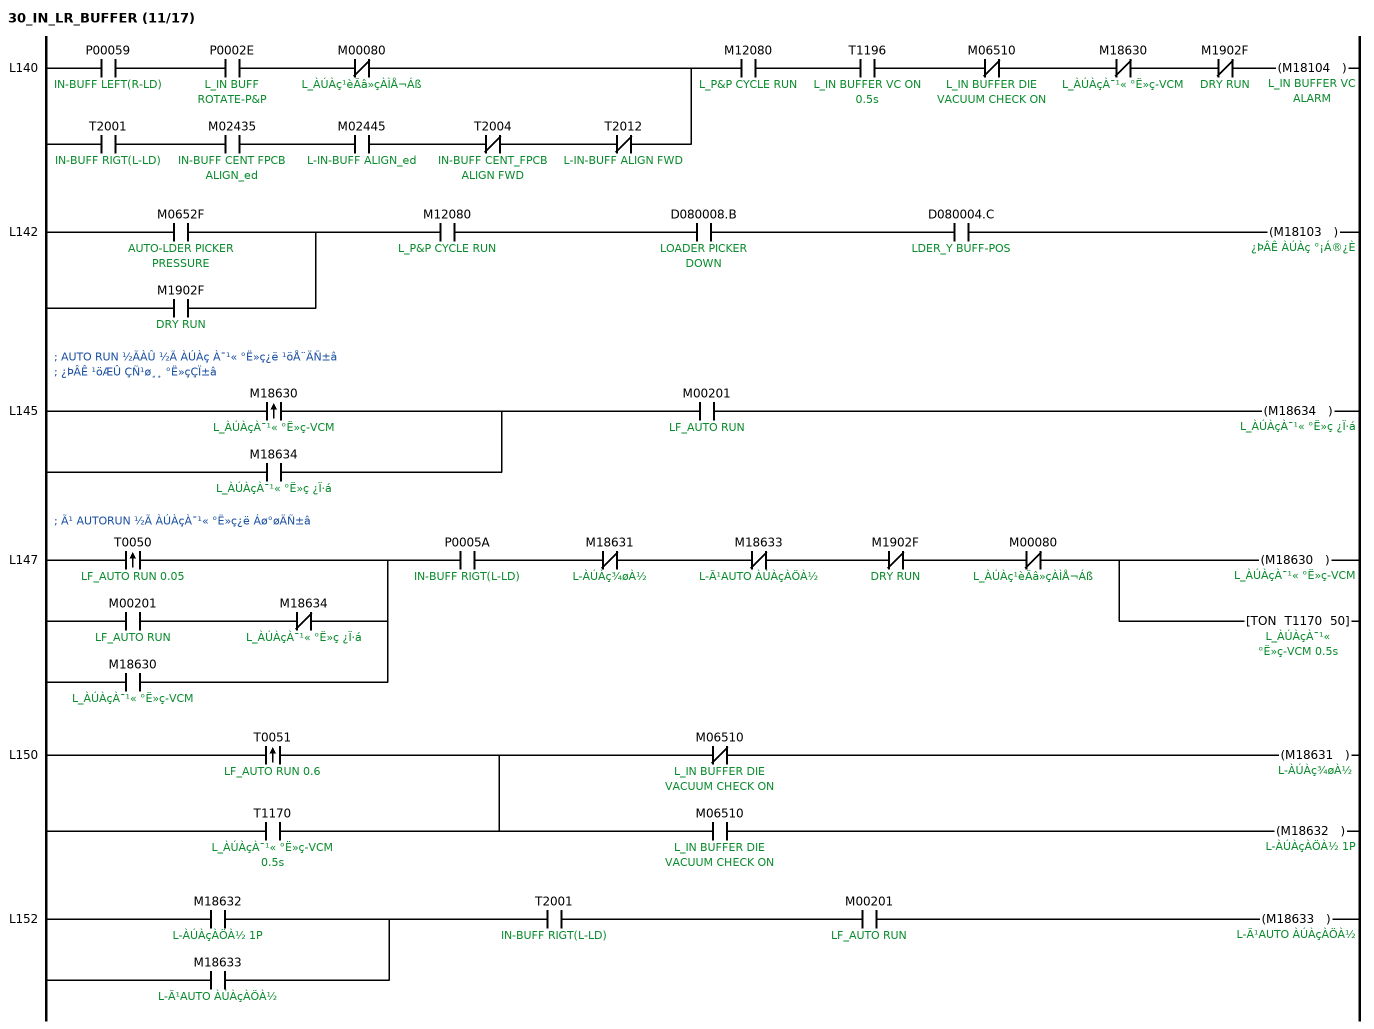
[picture p216: 30_IN_LR_BUFFER rungs L140-L152]
; L140
LOAD      P00059	// IN-BUFF LEFT(R-LD)
AND       P0002E	// L_IN BUFF ROTATE-P&P
AND NOT   M00080	// L_ÀÚÀç¹èÃâ»çÀÌÅ¬Áß
LOAD      T2001	// IN-BUFF RIGT(L-LD)
AND       M02435	// IN-BUFF CENT FPCB ALIGN_ed
AND       M02445	// L-IN-BUFF ALIGN_ed
AND NOT   T2004	// IN-BUFF CENT_FPCB ALIGN FWD
AND NOT   T2012	// L-IN-BUFF ALIGN FWD
OR LOAD
AND       M12080	// L_P&P CYCLE RUN
AND       T1196	// L_IN BUFFER VC ON 0.5s
AND NOT   M06510	// L_IN BUFFER DIE VACUUM CHECK ON
AND NOT   M18630	// L_ÀÚÀçÀ¯¹« °Ë»ç-VCM
AND NOT   M1902F	// DRY RUN
OUT       M18104	// L_IN BUFFER VC ALARM
; L142
LOAD      M0652F	// AUTO-LDER PICKER PRESSURE
OR        M1902F	// DRY RUN
AND       M12080	// L_P&P CYCLE RUN
AND       D080008.B	// LOADER PICKER DOWN
AND       D080004.C	// LDER_Y BUFF-POS
OUT       M18103	// ¿ÞÂÊ ÀÚÀç °¡Á®¿È
// AUTO RUN ½ÃÀÛ ½Ã ÀÚÀç À¯¹« °Ë»ç¿ë ¹öÅ¨ÄÑ±â
; L145
LOADP     M18630	// L_ÀÚÀçÀ¯¹« °Ë»ç-VCM
OR        M18634	// L_ÀÚÀçÀ¯¹« °Ë»ç ¿Ï·á
AND       M00201	// LF_AUTO RUN
OUT       M18634	// L_ÀÚÀçÀ¯¹« °Ë»ç ¿Ï·á
// output comment: ¿ÞÂÊ ¹öÆÛ ÇÑ¹ø¸¸ °Ë»çÇÏ±â
; L147
LOADP     T0050	// LF_AUTO RUN 0.05
LOAD      M00201	// LF_AUTO RUN
AND NOT   M18634	// L_ÀÚÀçÀ¯¹« °Ë»ç ¿Ï·á
OR LOAD
OR        M18630	// L_ÀÚÀçÀ¯¹« °Ë»ç-VCM
AND       P0005A	// IN-BUFF RIGT(L-LD)
AND NOT   M18631	// L-ÀÚÀç¾øÀ½
AND NOT   M18633	// L-Ã¹AUTO ÀÚÀçÀÖÀ½
AND NOT   M1902F	// DRY RUN
AND NOT   M00080	// L_ÀÚÀç¹èÃâ»çÀÌÅ¬Áß
OUT       M18630	// L_ÀÚÀçÀ¯¹« °Ë»ç-VCM
TON       T1170 50	// L_ÀÚÀçÀ¯¹« °Ë»ç-VCM 0.5s
// output comment: Ã¹ AUTORUN ½Ã ÀÚÀçÀ¯¹« °Ë»ç¿ë Áø°øÄÑ±â
; L150
LOADP     T0051	// LF_AUTO RUN 0.6
OR        T1170	// L_ÀÚÀçÀ¯¹« °Ë»ç-VCM 0.5s
MPUSH
AND NOT   M06510	// L_IN BUFFER DIE VACUUM CHECK ON
OUT       M18631	// L-ÀÚÀç¾øÀ½
MPOP
AND       M06510	// L_IN BUFFER DIE VACUUM CHECK ON
OUT       M18632	// L-ÀÚÀçÀÖÀ½ 1P
; L152
LOAD      M18632	// L-ÀÚÀçÀÖÀ½ 1P
OR        M18633	// L-Ã¹AUTO ÀÚÀçÀÖÀ½
AND       T2001	// IN-BUFF RIGT(L-LD)
AND       M00201	// LF_AUTO RUN
OUT       M18633	// L-Ã¹AUTO ÀÚÀçÀÖÀ½

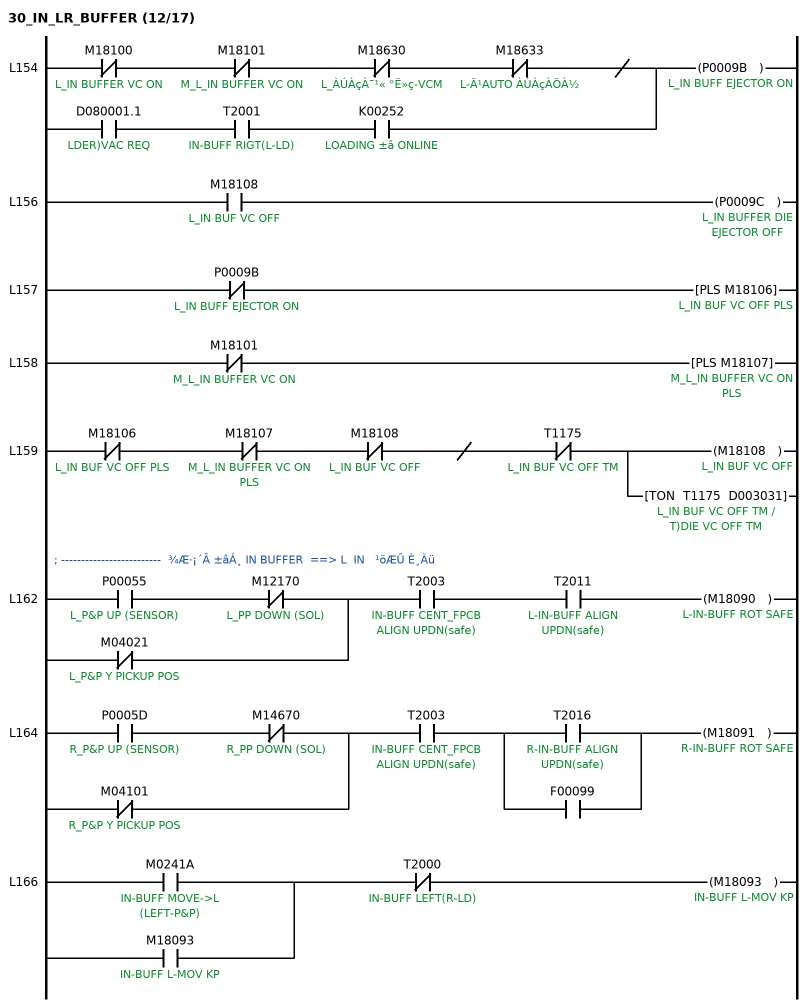
; L154
LOAD NOT  M18100	// L_IN BUFFER VC ON
AND NOT   M18101	// M_L_IN BUFFER VC ON
AND NOT   M18630	// L_ÀÚÀçÀ¯¹« °Ë»ç-VCM
AND NOT   M18633	// L-Ã¹AUTO ÀÚÀçÀÖÀ½
NOT
LOAD      D080001.1	// LDER)VAC REQ
AND       T2001	// IN-BUFF RIGT(L-LD)
AND       K00252	// LOADING ±â ONLINE
OR LOAD
OUT       P0009B	// L_IN BUFF EJECTOR ON
; L156
LOAD      M18108	// L_IN BUF VC OFF
OUT       P0009C	// L_IN BUFFER DIE EJECTOR OFF
; L157
LOAD NOT  P0009B	// L_IN BUFF EJECTOR ON
OUTP      M18106	// L_IN BUF VC OFF PLS
; L158
LOAD NOT  M18101	// M_L_IN BUFFER VC ON
OUTP      M18107	// M_L_IN BUFFER VC ON PLS
; L159
LOAD NOT  M18106	// L_IN BUF VC OFF PLS
AND NOT   M18107	// M_L_IN BUFFER VC ON PLS
AND NOT   M18108	// L_IN BUF VC OFF
NOT
AND NOT   T1175	// L_IN BUF VC OFF TM
OUT       M18108	// L_IN BUF VC OFF
TON       T1175 D003031	// L_IN BUF VC OFF TM / T)DIE VC OFF TM
// -------------------------  ¾Æ·¡´Â ±âÁ¸ IN BUFFER  ==> L  IN   ¹öÆÛ È¸Àü
; L162
LOAD      P00055	// L_P&P UP (SENSOR)
AND NOT   M12170	// L_PP DOWN (SOL)
OR NOT    M04021	// L_P&P Y PICKUP POS
AND       T2003	// IN-BUFF CENT_FPCB ALIGN UPDN(safe)
AND       T2011	// L-IN-BUFF ALIGN UPDN(safe)
OUT       M18090	// L-IN-BUFF ROT SAFE
; L164
LOAD      P0005D	// R_P&P UP (SENSOR)
AND NOT   M14670	// R_PP DOWN (SOL)
OR NOT    M04101	// R_P&P Y PICKUP POS
AND       T2003	// IN-BUFF CENT_FPCB ALIGN UPDN(safe)
LOAD      T2016	// R-IN-BUFF ALIGN UPDN(safe)
OR        F00099
AND LOAD
OUT       M18091	// R-IN-BUFF ROT SAFE
; L166
LOAD      M0241A	// IN-BUFF MOVE->L (LEFT-P&P)
OR        M18093	// IN-BUFF L-MOV KP
AND NOT   T2000	// IN-BUFF LEFT(R-LD)
OUT       M18093	// IN-BUFF L-MOV KP

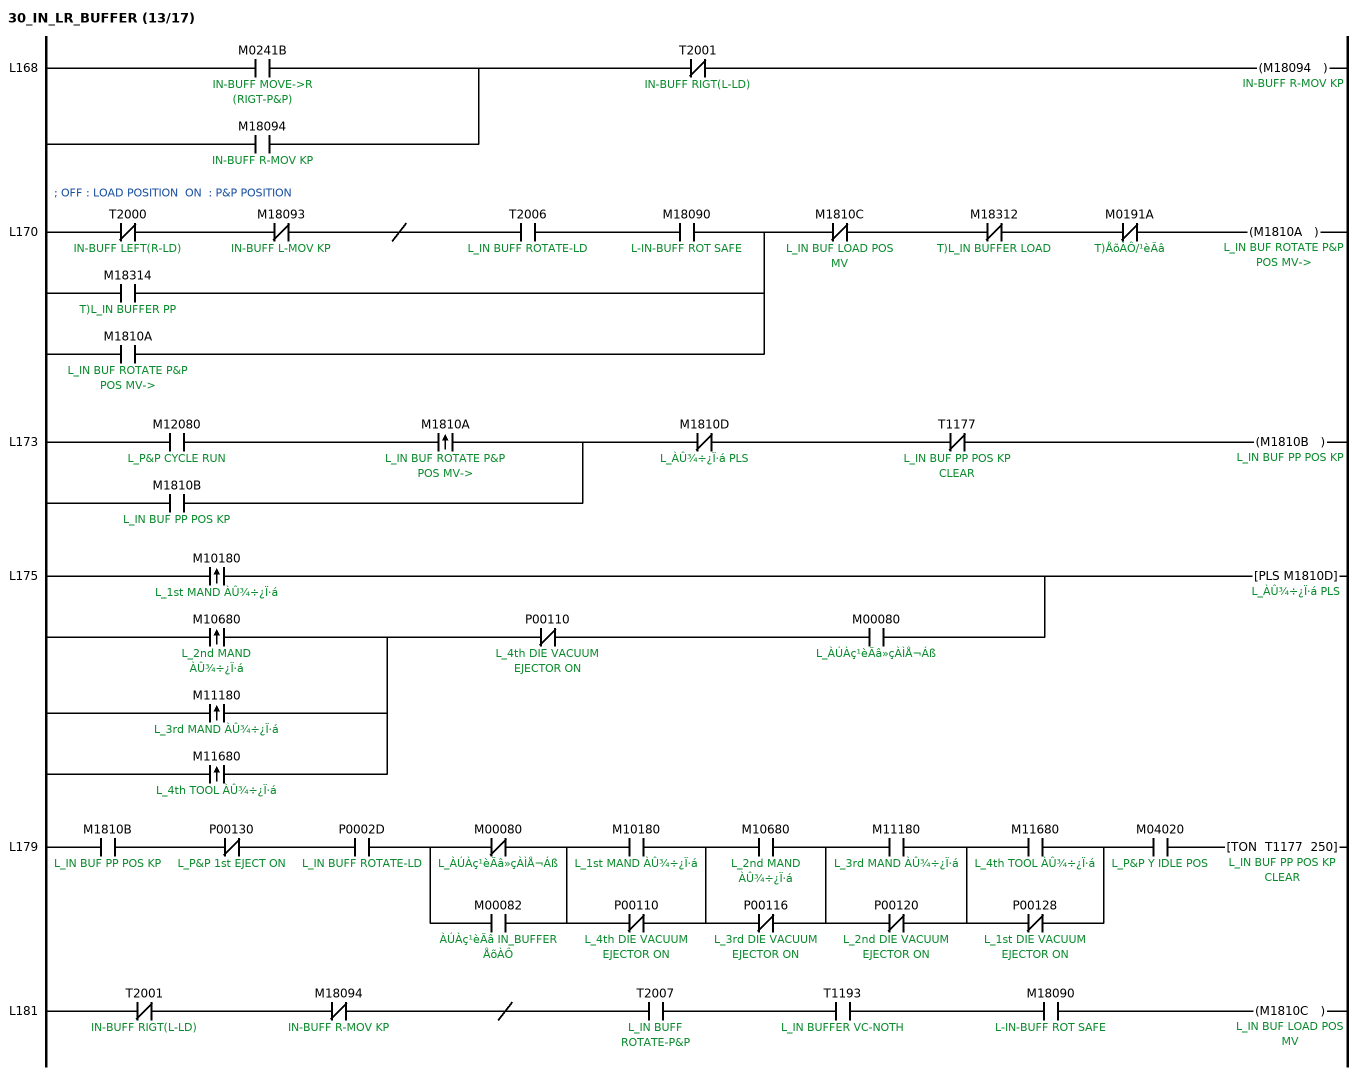
; L168
LOAD      M0241B	// IN-BUFF MOVE->R (RIGT-P&P)
OR        M18094	// IN-BUFF R-MOV KP
AND NOT   T2001	// IN-BUFF RIGT(L-LD)
OUT       M18094	// IN-BUFF R-MOV KP
; L170
LOAD NOT  T2000	// IN-BUFF LEFT(R-LD)
AND NOT   M18093	// IN-BUFF L-MOV KP
NOT
AND       T2006	// L_IN BUFF ROTATE-LD
AND       M18090	// L-IN-BUFF ROT SAFE
OR        M18314	// T)L_IN BUFFER PP
OR        M1810A	// L_IN BUF ROTATE P&P POS MV->
AND NOT   M1810C	// L_IN BUF LOAD POS MV
AND NOT   M18312	// T)L_IN BUFFER LOAD
AND NOT   M0191A	// T)ÅõÀÔ/¹èÃâ
OUT       M1810A	// L_IN BUF ROTATE P&P POS MV->
// output comment: OFF : LOAD POSITION  ON  : P&P POSITION
; L173
LOAD      M12080	// L_P&P CYCLE RUN
ANDP      M1810A	// L_IN BUF ROTATE P&P POS MV->
OR        M1810B	// L_IN BUF PP POS KP
AND NOT   M1810D	// L_ÀÛ¾÷¿Ï·á PLS
AND NOT   T1177	// L_IN BUF PP POS KP CLEAR
OUT       M1810B	// L_IN BUF PP POS KP
; L175
LOADP     M10180	// L_1st MAND ÀÛ¾÷¿Ï·á
LOADP     M10680	// L_2nd MAND ÀÛ¾÷¿Ï·á
ORP       M11180	// L_3rd MAND ÀÛ¾÷¿Ï·á
ORP       M11680	// L_4th TOOL ÀÛ¾÷¿Ï·á
AND NOT   P00110	// L_4th DIE VACUUM EJECTOR ON
AND       M00080	// L_ÀÚÀç¹èÃâ»çÀÌÅ¬Áß
OR LOAD
OUTP      M1810D	// L_ÀÛ¾÷¿Ï·á PLS
; L179
LOAD      M1810B	// L_IN BUF PP POS KP
AND NOT   P00130	// L_P&P 1st EJECT ON
AND       P0002D	// L_IN BUFF ROTATE-LD
LOAD NOT  M00080	// L_ÀÚÀç¹èÃâ»çÀÌÅ¬Áß
OR        M00082	// ÀÚÀç¹èÃâ IN_BUFFER ÅõÀÔ 
AND LOAD
LOAD      M10180	// L_1st MAND ÀÛ¾÷¿Ï·á
OR NOT    P00110	// L_4th DIE VACUUM EJECTOR ON
AND LOAD
LOAD      M10680	// L_2nd MAND ÀÛ¾÷¿Ï·á
OR NOT    P00116	// L_3rd DIE VACUUM EJECTOR ON
AND LOAD
LOAD      M11180	// L_3rd MAND ÀÛ¾÷¿Ï·á
OR NOT    P00120	// L_2nd DIE VACUUM EJECTOR ON
AND LOAD
LOAD      M11680	// L_4th TOOL ÀÛ¾÷¿Ï·á
OR NOT    P00128	// L_1st DIE VACUUM EJECTOR ON
AND LOAD
AND       M04020	// L_P&P Y IDLE POS
TON       T1177 250	// L_IN BUF PP POS KP CLEAR
; L181
LOAD NOT  T2001	// IN-BUFF RIGT(L-LD)
AND NOT   M18094	// IN-BUFF R-MOV KP
NOT
AND       T2007	// L_IN BUFF ROTATE-P&P
AND       T1193	// L_IN BUFFER VC-NOTH
AND       M18090	// L-IN-BUFF ROT SAFE
OUT       M1810C	// L_IN BUF LOAD POS MV

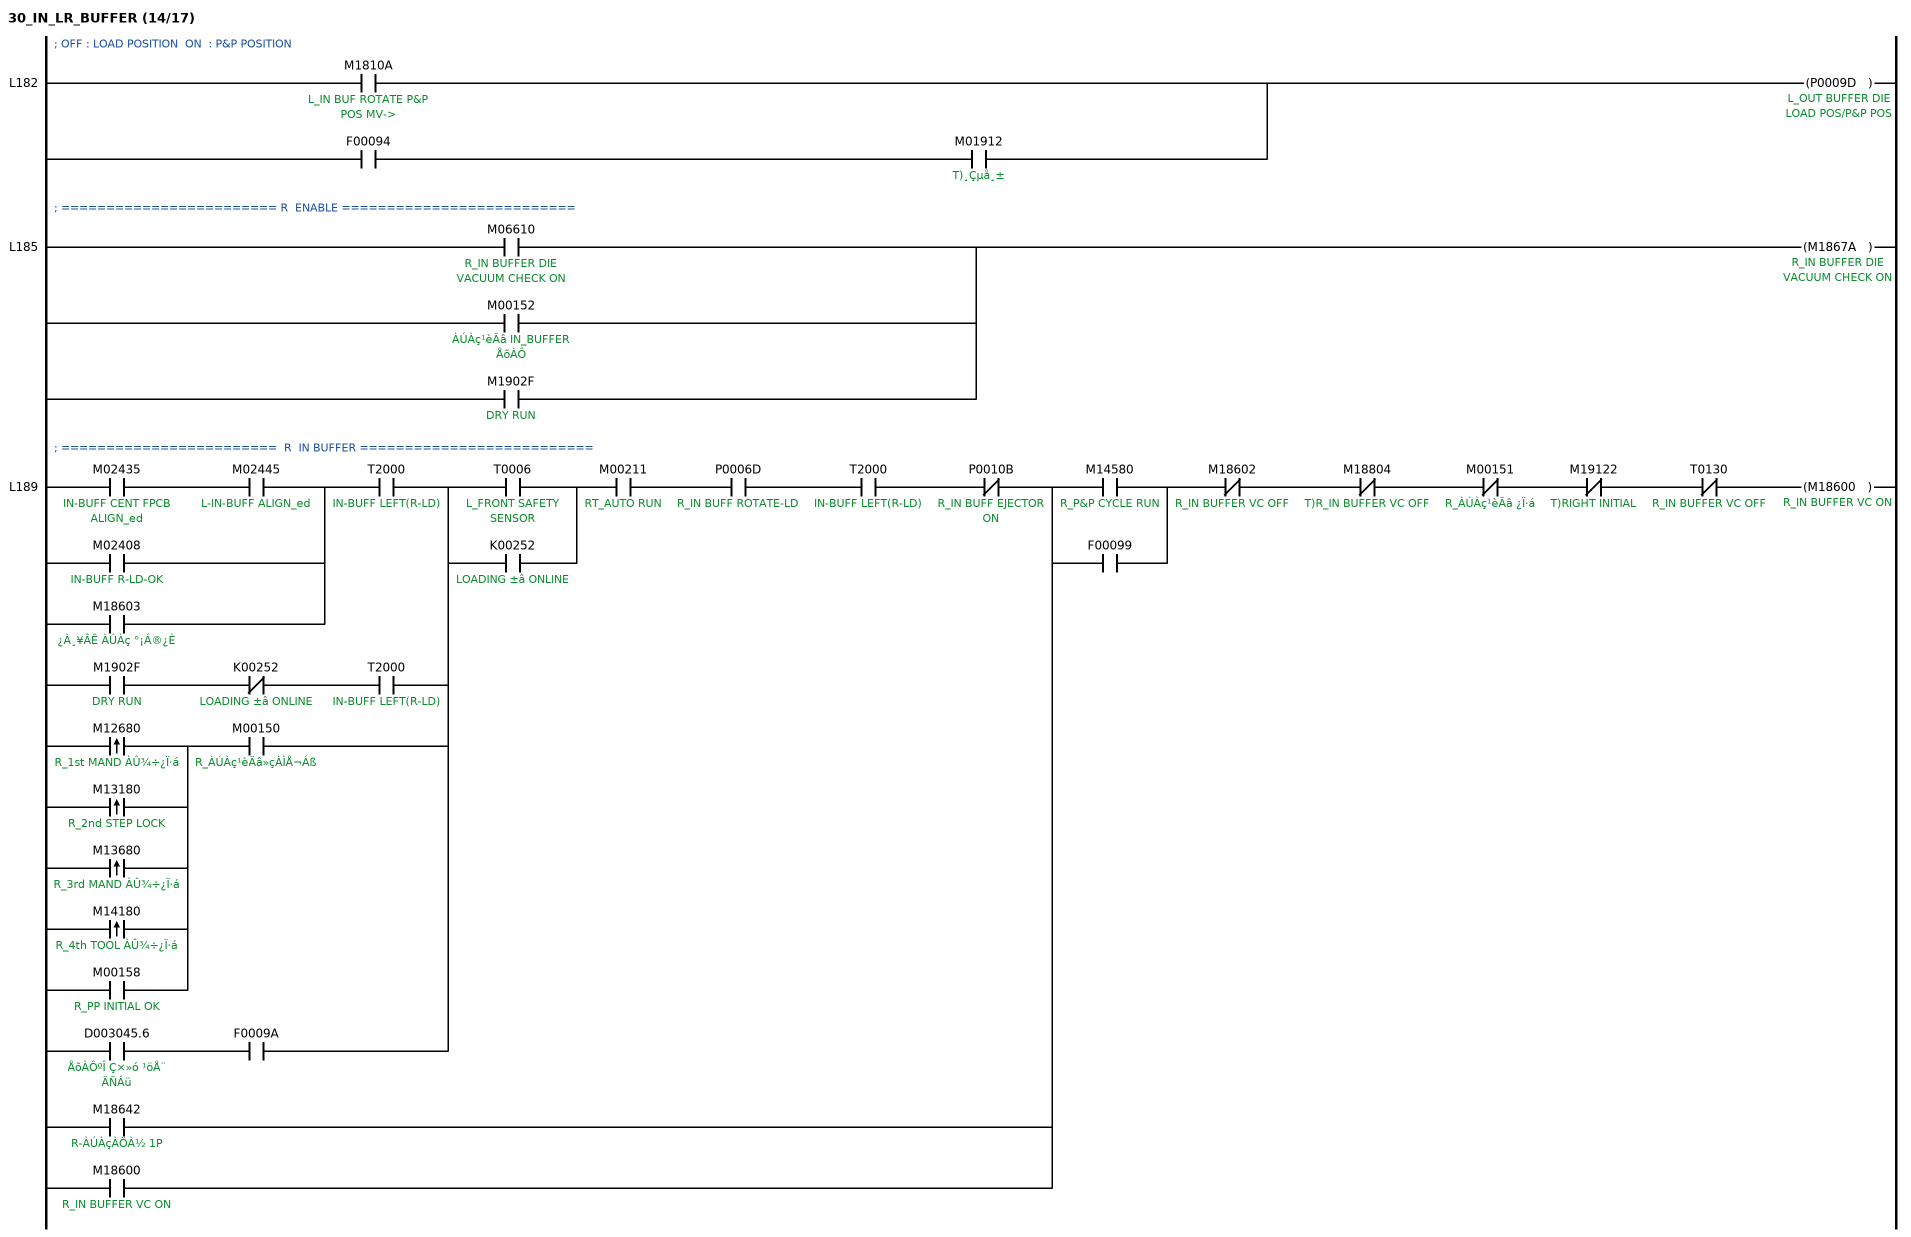
; L182
LOAD      M1810A	// L_IN BUF ROTATE P&P POS MV->
LOAD      F00094
AND       M01912	// T)¸Çµå¸±
OR LOAD
OUT       P0009D	// L_OUT BUFFER DIE LOAD POS/P&P POS
// output comment: OFF : LOAD POSITION  ON  : P&P POSITION
// ======================== R  ENABLE ==========================
; L185
LOAD      M06610	// R_IN BUFFER DIE VACUUM CHECK ON
OR        M00152	// ÀÚÀç¹èÃâ IN_BUFFER ÅõÀÔ 
OR        M1902F	// DRY RUN
OUT       M1867A	// R_IN BUFFER DIE VACUUM CHECK ON
// ========================  R  IN BUFFER ==========================
; L189
LOAD      M02435	// IN-BUFF CENT FPCB ALIGN_ed
AND       M02445	// L-IN-BUFF ALIGN_ed
OR        M02408	// IN-BUFF R-LD-OK
OR        M18603	// ¿À¸¥ÂÊ ÀÚÀç °¡Á®¿È
AND       T2000	// IN-BUFF LEFT(R-LD)
LOAD      M1902F	// DRY RUN
AND NOT   K00252	// LOADING ±â ONLINE
AND       T2000	// IN-BUFF LEFT(R-LD)
OR LOAD
LOADP     M12680	// R_1st MAND ÀÛ¾÷¿Ï·á
ORP       M13180	// R_2nd STEP LOCK
ORP       M13680	// R_3rd MAND ÀÛ¾÷¿Ï·á
ORP       M14180	// R_4th TOOL ÀÛ¾÷¿Ï·á
OR        M00158	// R_PP INITIAL OK
AND       M00150	// R_ÀÚÀç¹èÃâ»çÀÌÅ¬Áß
OR LOAD
LOAD      D003045.6	// ÅõÀÔºÎ Ç×»ó ¹öÅ¨ ÄÑÁü
AND       F0009A
OR LOAD
LOAD      T0006	// L_FRONT SAFETY SENSOR
OR        K00252	// LOADING ±â ONLINE
AND LOAD
AND       M00211	// RT_AUTO RUN
AND       P0006D	// R_IN BUFF ROTATE-LD
AND       T2000	// IN-BUFF LEFT(R-LD)
AND NOT   P0010B	// R_IN BUFF EJECTOR ON
OR        M18642	// R-ÀÚÀçÀÖÀ½ 1P
OR        M18600	// R_IN BUFFER VC ON
LOAD      M14580	// R_P&P CYCLE RUN
OR        F00099
AND LOAD
AND NOT   M18602	// R_IN BUFFER VC OFF
AND NOT   M18804	// T)R_IN BUFFER VC OFF
AND NOT   M00151	// R_ÀÚÀç¹èÃâ ¿Ï·á
AND NOT   M19122	// T)RIGHT INITIAL
AND NOT   T0130	// R_IN BUFFER VC OFF
OUT       M18600	// R_IN BUFFER VC ON

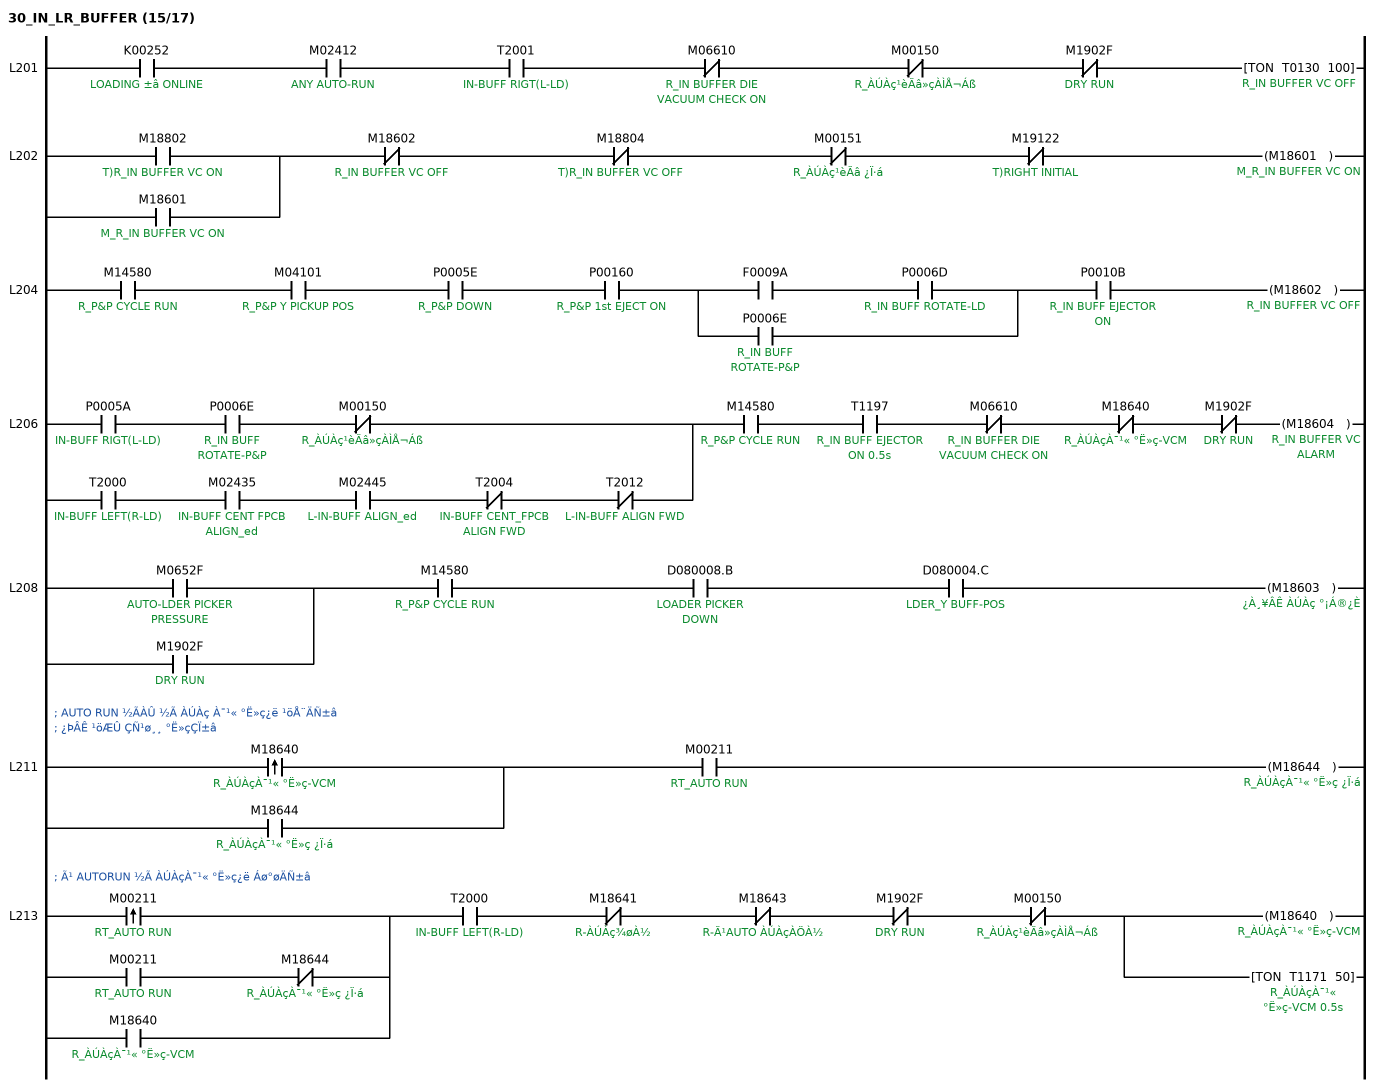
; L201
LOAD      K00252	// LOADING ±â ONLINE
AND       M02412	// ANY AUTO-RUN
AND       T2001	// IN-BUFF RIGT(L-LD)
AND NOT   M06610	// R_IN BUFFER DIE VACUUM CHECK ON
AND NOT   M00150	// R_ÀÚÀç¹èÃâ»çÀÌÅ¬Áß
AND NOT   M1902F	// DRY RUN
TON       T0130 100	// R_IN BUFFER VC OFF
; L202
LOAD      M18802	// T)R_IN BUFFER VC ON
OR        M18601	// M_R_IN BUFFER VC ON
AND NOT   M18602	// R_IN BUFFER VC OFF
AND NOT   M18804	// T)R_IN BUFFER VC OFF
AND NOT   M00151	// R_ÀÚÀç¹èÃâ ¿Ï·á
AND NOT   M19122	// T)RIGHT INITIAL
OUT       M18601	// M_R_IN BUFFER VC ON
; L204
LOAD      M14580	// R_P&P CYCLE RUN
AND       M04101	// R_P&P Y PICKUP POS
AND       P0005E	// R_P&P DOWN
AND       P00160	// R_P&P 1st EJECT ON
LOAD      F0009A
AND       P0006D	// R_IN BUFF ROTATE-LD
OR        P0006E	// R_IN BUFF ROTATE-P&P
AND LOAD
AND       P0010B	// R_IN BUFF EJECTOR ON
OUT       M18602	// R_IN BUFFER VC OFF
; L206
LOAD      P0005A	// IN-BUFF RIGT(L-LD)
AND       P0006E	// R_IN BUFF ROTATE-P&P
AND NOT   M00150	// R_ÀÚÀç¹èÃâ»çÀÌÅ¬Áß
LOAD      T2000	// IN-BUFF LEFT(R-LD)
AND       M02435	// IN-BUFF CENT FPCB ALIGN_ed
AND       M02445	// L-IN-BUFF ALIGN_ed
AND NOT   T2004	// IN-BUFF CENT_FPCB ALIGN FWD
AND NOT   T2012	// L-IN-BUFF ALIGN FWD
OR LOAD
AND       M14580	// R_P&P CYCLE RUN
AND       T1197	// R_IN BUFF EJECTOR ON 0.5s
AND NOT   M06610	// R_IN BUFFER DIE VACUUM CHECK ON
AND NOT   M18640	// R_ÀÚÀçÀ¯¹« °Ë»ç-VCM
AND NOT   M1902F	// DRY RUN
OUT       M18604	// R_IN BUFFER VC ALARM
; L208
LOAD      M0652F	// AUTO-LDER PICKER PRESSURE
OR        M1902F	// DRY RUN
AND       M14580	// R_P&P CYCLE RUN
AND       D080008.B	// LOADER PICKER DOWN
AND       D080004.C	// LDER_Y BUFF-POS
OUT       M18603	// ¿À¸¥ÂÊ ÀÚÀç °¡Á®¿È
// AUTO RUN ½ÃÀÛ ½Ã ÀÚÀç À¯¹« °Ë»ç¿ë ¹öÅ¨ÄÑ±â
; L211
LOADP     M18640	// R_ÀÚÀçÀ¯¹« °Ë»ç-VCM
OR        M18644	// R_ÀÚÀçÀ¯¹« °Ë»ç ¿Ï·á
AND       M00211	// RT_AUTO RUN
OUT       M18644	// R_ÀÚÀçÀ¯¹« °Ë»ç ¿Ï·á
// output comment: ¿ÞÂÊ ¹öÆÛ ÇÑ¹ø¸¸ °Ë»çÇÏ±â
; L213
LOADP     M00211	// RT_AUTO RUN
LOAD      M00211	// RT_AUTO RUN
AND NOT   M18644	// R_ÀÚÀçÀ¯¹« °Ë»ç ¿Ï·á
OR LOAD
OR        M18640	// R_ÀÚÀçÀ¯¹« °Ë»ç-VCM
AND       T2000	// IN-BUFF LEFT(R-LD)
AND NOT   M18641	// R-ÀÚÀç¾øÀ½
AND NOT   M18643	// R-Ã¹AUTO ÀÚÀçÀÖÀ½
AND NOT   M1902F	// DRY RUN
AND NOT   M00150	// R_ÀÚÀç¹èÃâ»çÀÌÅ¬Áß
OUT       M18640	// R_ÀÚÀçÀ¯¹« °Ë»ç-VCM
TON       T1171 50	// R_ÀÚÀçÀ¯¹« °Ë»ç-VCM 0.5s
// output comment: Ã¹ AUTORUN ½Ã ÀÚÀçÀ¯¹« °Ë»ç¿ë Áø°øÄÑ±â

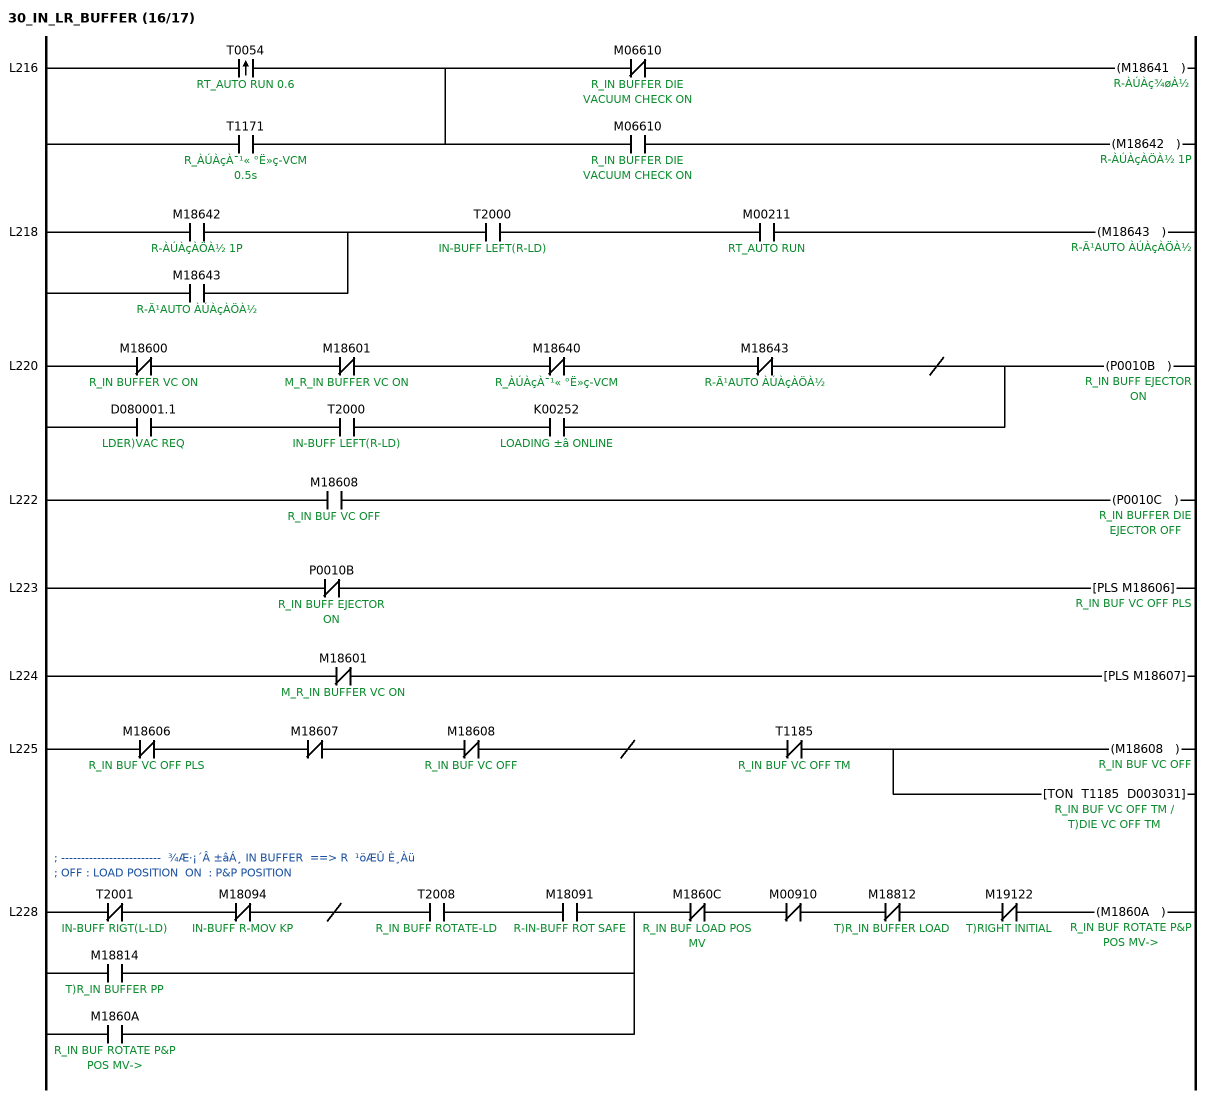
; L216
LOADP     T0054	// RT_AUTO RUN 0.6
OR        T1171	// R_ÀÚÀçÀ¯¹« °Ë»ç-VCM 0.5s
MPUSH
AND NOT   M06610	// R_IN BUFFER DIE VACUUM CHECK ON
OUT       M18641	// R-ÀÚÀç¾øÀ½
MPOP
AND       M06610	// R_IN BUFFER DIE VACUUM CHECK ON
OUT       M18642	// R-ÀÚÀçÀÖÀ½ 1P
; L218
LOAD      M18642	// R-ÀÚÀçÀÖÀ½ 1P
OR        M18643	// R-Ã¹AUTO ÀÚÀçÀÖÀ½
AND       T2000	// IN-BUFF LEFT(R-LD)
AND       M00211	// RT_AUTO RUN
OUT       M18643	// R-Ã¹AUTO ÀÚÀçÀÖÀ½
; L220
LOAD NOT  M18600	// R_IN BUFFER VC ON
AND NOT   M18601	// M_R_IN BUFFER VC ON
AND NOT   M18640	// R_ÀÚÀçÀ¯¹« °Ë»ç-VCM
AND NOT   M18643	// R-Ã¹AUTO ÀÚÀçÀÖÀ½
NOT
LOAD      D080001.1	// LDER)VAC REQ
AND       T2000	// IN-BUFF LEFT(R-LD)
AND       K00252	// LOADING ±â ONLINE
OR LOAD
OUT       P0010B	// R_IN BUFF EJECTOR ON
; L222
LOAD      M18608	// R_IN BUF VC OFF
OUT       P0010C	// R_IN BUFFER DIE EJECTOR OFF
; L223
LOAD NOT  P0010B	// R_IN BUFF EJECTOR ON
OUTP      M18606	// R_IN BUF VC OFF PLS
; L224
LOAD NOT  M18601	// M_R_IN BUFFER VC ON
OUTP      M18607
; L225
LOAD NOT  M18606	// R_IN BUF VC OFF PLS
AND NOT   M18607
AND NOT   M18608	// R_IN BUF VC OFF
NOT
AND NOT   T1185	// R_IN BUF VC OFF TM
OUT       M18608	// R_IN BUF VC OFF
TON       T1185 D003031	// R_IN BUF VC OFF TM / T)DIE VC OFF TM
// -------------------------  ¾Æ·¡´Â ±âÁ¸ IN BUFFER  ==> R  ¹öÆÛ È¸Àü
; L228
LOAD NOT  T2001	// IN-BUFF RIGT(L-LD)
AND NOT   M18094	// IN-BUFF R-MOV KP
NOT
AND       T2008	// R_IN BUFF ROTATE-LD
AND       M18091	// R-IN-BUFF ROT SAFE
OR        M18814	// T)R_IN BUFFER PP
OR        M1860A	// R_IN BUF ROTATE P&P POS MV->
AND NOT   M1860C	// R_IN BUF LOAD POS MV
AND NOT   M00910
AND NOT   M18812	// T)R_IN BUFFER LOAD
AND NOT   M19122	// T)RIGHT INITIAL
OUT       M1860A	// R_IN BUF ROTATE P&P POS MV->
// output comment: OFF : LOAD POSITION  ON  : P&P POSITION

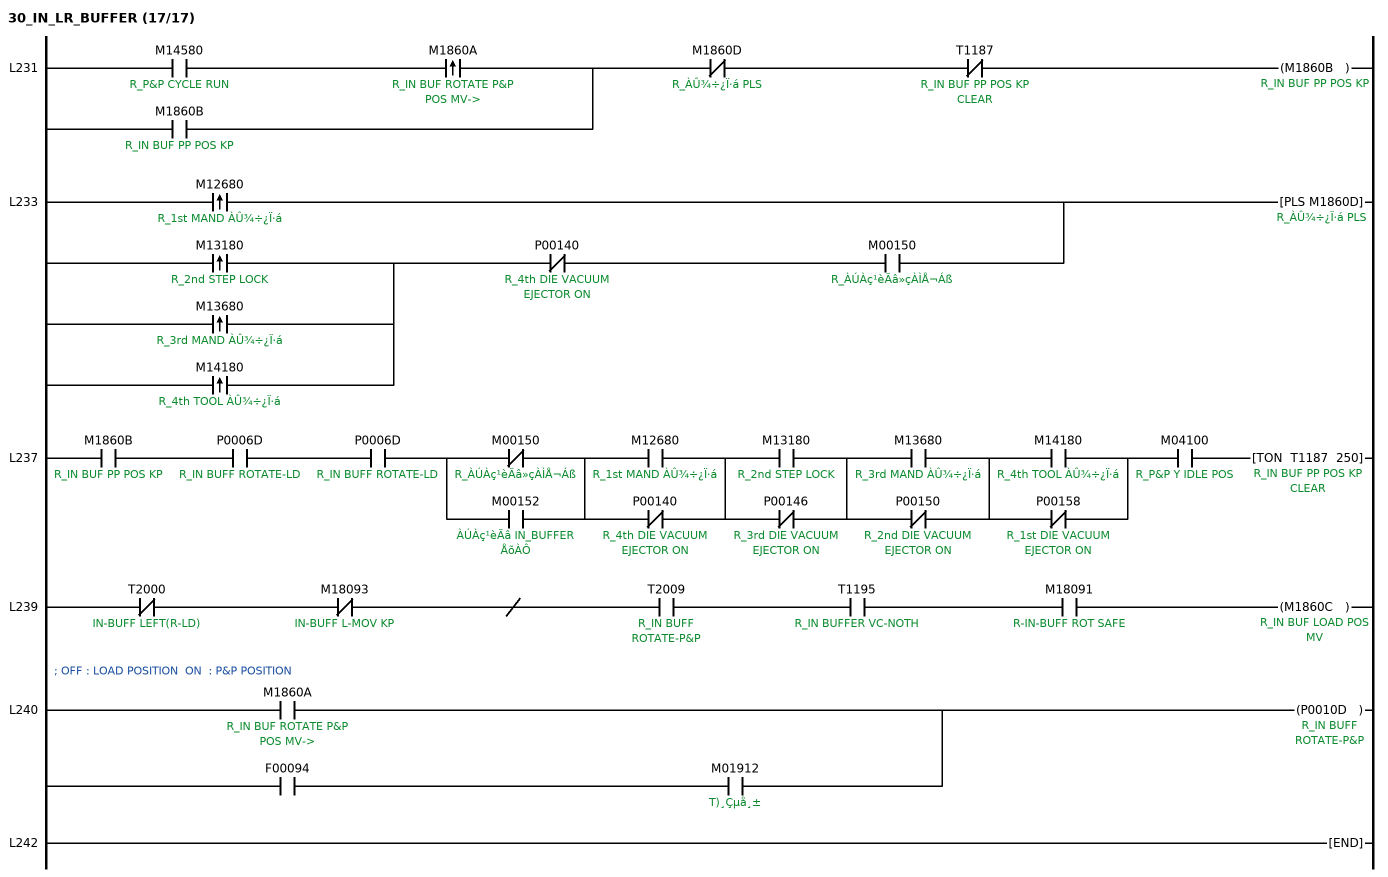
; L231
LOAD      M14580	// R_P&P CYCLE RUN
ANDP      M1860A	// R_IN BUF ROTATE P&P POS MV->
OR        M1860B	// R_IN BUF PP POS KP
AND NOT   M1860D	// R_ÀÛ¾÷¿Ï·á PLS
AND NOT   T1187	// R_IN BUF PP POS KP CLEAR
OUT       M1860B	// R_IN BUF PP POS KP
; L233
LOADP     M12680	// R_1st MAND ÀÛ¾÷¿Ï·á
LOADP     M13180	// R_2nd STEP LOCK
ORP       M13680	// R_3rd MAND ÀÛ¾÷¿Ï·á
ORP       M14180	// R_4th TOOL ÀÛ¾÷¿Ï·á
AND NOT   P00140	// R_4th DIE VACUUM EJECTOR ON
AND       M00150	// R_ÀÚÀç¹èÃâ»çÀÌÅ¬Áß
OR LOAD
OUTP      M1860D	// R_ÀÛ¾÷¿Ï·á PLS
; L237
LOAD      M1860B	// R_IN BUF PP POS KP
AND       P0006D	// R_IN BUFF ROTATE-LD
AND       P0006D	// R_IN BUFF ROTATE-LD
LOAD NOT  M00150	// R_ÀÚÀç¹èÃâ»çÀÌÅ¬Áß
OR        M00152	// ÀÚÀç¹èÃâ IN_BUFFER ÅõÀÔ 
AND LOAD
LOAD      M12680	// R_1st MAND ÀÛ¾÷¿Ï·á
OR NOT    P00140	// R_4th DIE VACUUM EJECTOR ON
AND LOAD
LOAD      M13180	// R_2nd STEP LOCK
OR NOT    P00146	// R_3rd DIE VACUUM EJECTOR ON
AND LOAD
LOAD      M13680	// R_3rd MAND ÀÛ¾÷¿Ï·á
OR NOT    P00150	// R_2nd DIE VACUUM EJECTOR ON
AND LOAD
LOAD      M14180	// R_4th TOOL ÀÛ¾÷¿Ï·á
OR NOT    P00158	// R_1st DIE VACUUM EJECTOR ON
AND LOAD
AND       M04100	// R_P&P Y IDLE POS
TON       T1187 250	// R_IN BUF PP POS KP CLEAR
; L239
LOAD NOT  T2000	// IN-BUFF LEFT(R-LD)
AND NOT   M18093	// IN-BUFF L-MOV KP
NOT
AND       T2009	// R_IN BUFF ROTATE-P&P
AND       T1195	// R_IN BUFFER VC-NOTH
AND       M18091	// R-IN-BUFF ROT SAFE
OUT       M1860C	// R_IN BUF LOAD POS MV
; L240
LOAD      M1860A	// R_IN BUF ROTATE P&P POS MV->
LOAD      F00094
AND       M01912	// T)¸Çµå¸±
OR LOAD
OUT       P0010D	// R_IN BUFF ROTATE-P&P
// output comment: OFF : LOAD POSITION  ON  : P&P POSITION
; L242
END

PROGRAM 31_OUT_LR_BUFFER (task: ½ºÄµ ÇÁ·Î±×·¥)

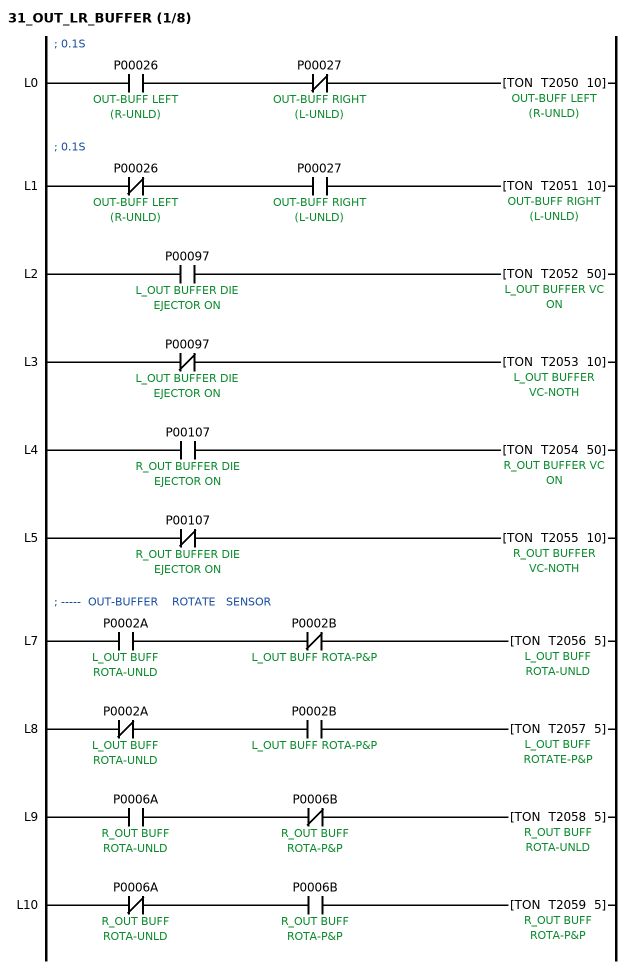
; L0
LOAD      P00026	// OUT-BUFF LEFT (R-UNLD)
AND NOT   P00027	// OUT-BUFF RIGHT (L-UNLD)
TON       T2050 10	// OUT-BUFF LEFT (R-UNLD)
// output comment: 0.1S
; L1
LOAD NOT  P00026	// OUT-BUFF LEFT (R-UNLD)
AND       P00027	// OUT-BUFF RIGHT (L-UNLD)
TON       T2051 10	// OUT-BUFF RIGHT (L-UNLD)
// output comment: 0.1S
; L2
LOAD      P00097	// L_OUT BUFFER DIE EJECTOR ON
TON       T2052 50	// L_OUT BUFFER VC ON
; L3
LOAD NOT  P00097	// L_OUT BUFFER DIE EJECTOR ON
TON       T2053 10	// L_OUT BUFFER VC-NOTH
; L4
LOAD      P00107	// R_OUT BUFFER DIE EJECTOR ON
TON       T2054 50	// R_OUT BUFFER VC ON
; L5
LOAD NOT  P00107	// R_OUT BUFFER DIE EJECTOR ON
TON       T2055 10	// R_OUT BUFFER VC-NOTH
// -----  OUT-BUFFER    ROTATE   SENSOR
; L7
LOAD      P0002A	// L_OUT BUFF ROTA-UNLD
AND NOT   P0002B	// L_OUT BUFF ROTA-P&P
TON       T2056 5	// L_OUT BUFF ROTA-UNLD
; L8
LOAD NOT  P0002A	// L_OUT BUFF ROTA-UNLD
AND       P0002B	// L_OUT BUFF ROTA-P&P
TON       T2057 5	// L_OUT BUFF ROTATE-P&P
; L9
LOAD      P0006A	// R_OUT BUFF ROTA-UNLD
AND NOT   P0006B	// R_OUT BUFF ROTA-P&P
TON       T2058 5	// R_OUT BUFF ROTA-UNLD
; L10
LOAD NOT  P0006A	// R_OUT BUFF ROTA-UNLD
AND       P0006B	// R_OUT BUFF ROTA-P&P
TON       T2059 5	// R_OUT BUFF ROTA-P&P

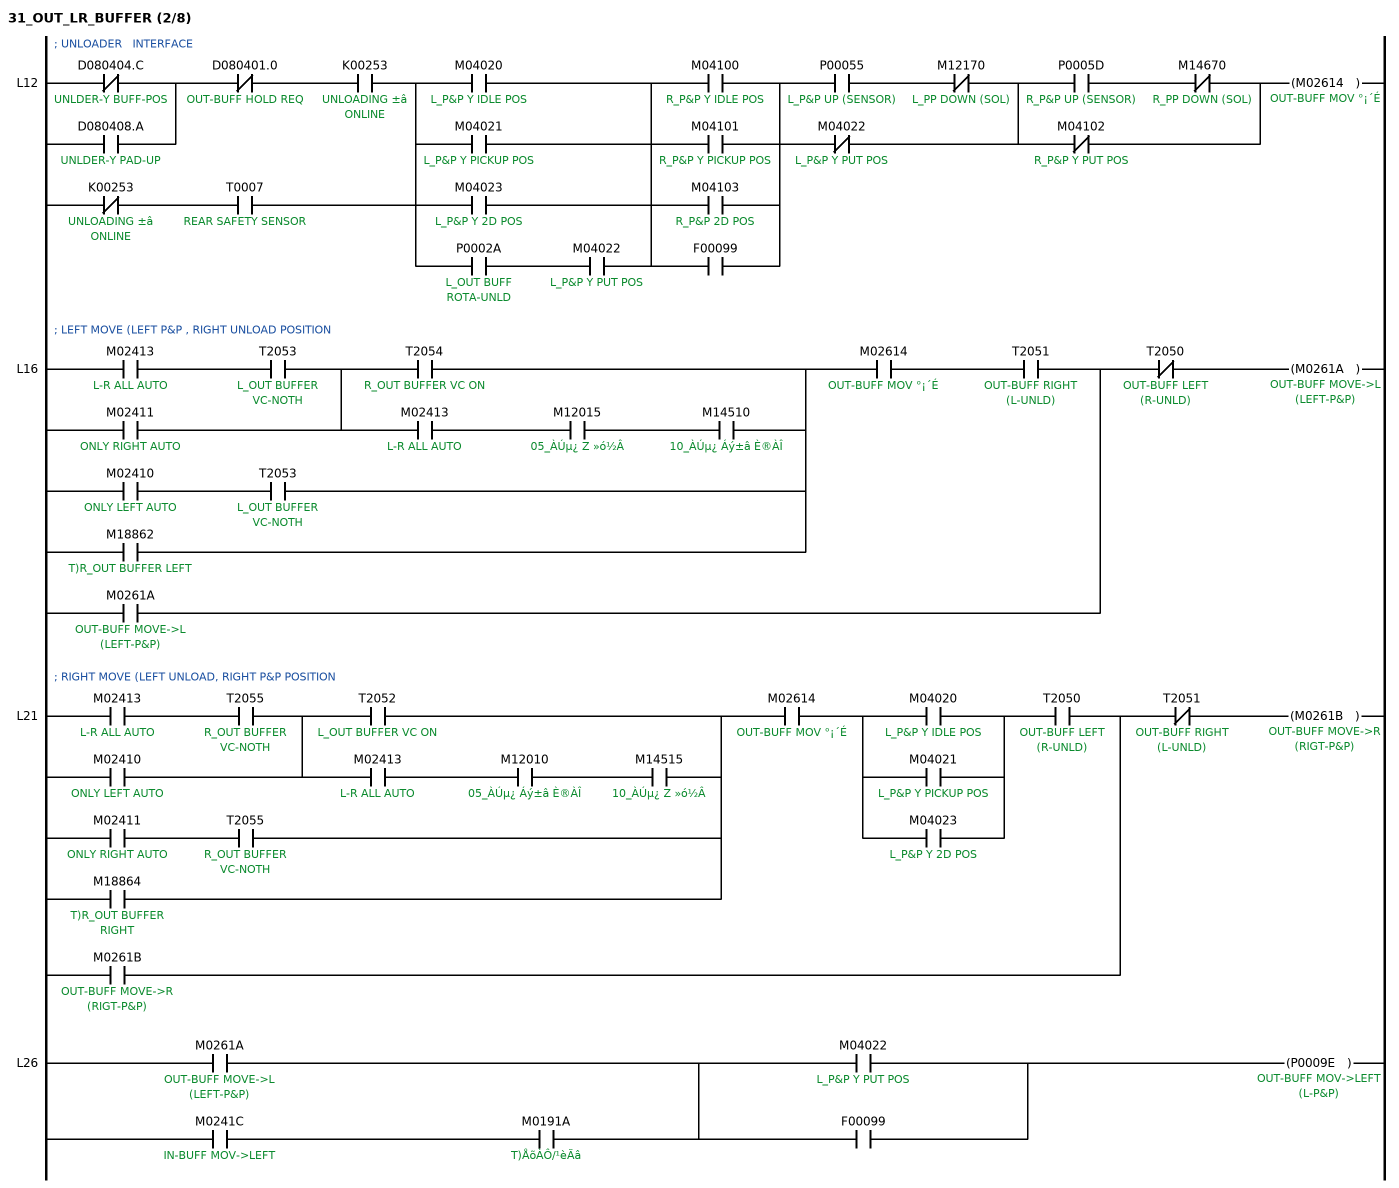
//  UNLOADER   INTERFACE
; L12
LOAD NOT  D080404.C	// UNLDER-Y BUFF-POS
OR        D080408.A	// UNLDER-Y PAD-UP
AND NOT   D080401.0	// OUT-BUFF HOLD REQ
AND       K00253	// UNLOADING ±â ONLINE
LOAD NOT  K00253	// UNLOADING ±â ONLINE
AND       T0007	// REAR SAFETY SENSOR
OR LOAD
LOAD      M04020	// L_P&P Y IDLE POS
OR        M04021	// L_P&P Y PICKUP POS
OR        M04023	// L_P&P Y 2D POS
LOAD      P0002A	// L_OUT BUFF ROTA-UNLD
AND       M04022	// L_P&P Y PUT POS
OR LOAD
AND LOAD
LOAD      M04100	// R_P&P Y IDLE POS
OR        M04101	// R_P&P Y PICKUP POS
OR        M04103	// R_P&P 2D POS
OR        F00099
AND LOAD
LOAD      P00055	// L_P&P UP (SENSOR)
AND NOT   M12170	// L_PP DOWN (SOL)
OR NOT    M04022	// L_P&P Y PUT POS
AND LOAD
LOAD      P0005D	// R_P&P UP (SENSOR)
AND NOT   M14670	// R_PP DOWN (SOL)
OR NOT    M04102	// R_P&P Y PUT POS
AND LOAD
OUT       M02614	// OUT-BUFF MOV °¡´É
; L16
LOAD      M02413	// L-R ALL AUTO
AND       T2053	// L_OUT BUFFER VC-NOTH
OR        M02411	// ONLY RIGHT AUTO
LOAD      T2054	// R_OUT BUFFER VC ON
LOAD      M02413	// L-R ALL AUTO
AND       M12015	// 05_ÀÚµ¿ Z »ó½Â
AND       M14510	// 10_ÀÚµ¿ Áý±â È®ÀÎ
OR LOAD
AND LOAD
LOAD      M02410	// ONLY LEFT AUTO
AND       T2053	// L_OUT BUFFER VC-NOTH
OR LOAD
OR        M18862	// T)R_OUT BUFFER LEFT
AND       M02614	// OUT-BUFF MOV °¡´É
AND       T2051	// OUT-BUFF RIGHT (L-UNLD)
OR        M0261A	// OUT-BUFF MOVE->L (LEFT-P&P)
AND NOT   T2050	// OUT-BUFF LEFT (R-UNLD)
OUT       M0261A	// OUT-BUFF MOVE->L (LEFT-P&P)
// output comment: LEFT MOVE (LEFT P&P , RIGHT UNLOAD POSITION
; L21
LOAD      M02413	// L-R ALL AUTO
AND       T2055	// R_OUT BUFFER VC-NOTH
OR        M02410	// ONLY LEFT AUTO
LOAD      T2052	// L_OUT BUFFER VC ON
LOAD      M02413	// L-R ALL AUTO
AND       M12010	// 05_ÀÚµ¿ Áý±â È®ÀÎ
AND       M14515	// 10_ÀÚµ¿ Z »ó½Â
OR LOAD
AND LOAD
LOAD      M02411	// ONLY RIGHT AUTO
AND       T2055	// R_OUT BUFFER VC-NOTH
OR LOAD
OR        M18864	// T)R_OUT BUFFER RIGHT
AND       M02614	// OUT-BUFF MOV °¡´É
LOAD      M04020	// L_P&P Y IDLE POS
OR        M04021	// L_P&P Y PICKUP POS
OR        M04023	// L_P&P Y 2D POS
AND LOAD
AND       T2050	// OUT-BUFF LEFT (R-UNLD)
OR        M0261B	// OUT-BUFF MOVE->R (RIGT-P&P)
AND NOT   T2051	// OUT-BUFF RIGHT (L-UNLD)
OUT       M0261B	// OUT-BUFF MOVE->R (RIGT-P&P)
// output comment: RIGHT MOVE (LEFT UNLOAD, RIGHT P&P POSITION
; L26
LOAD      M0261A	// OUT-BUFF MOVE->L (LEFT-P&P)
LOAD      M0241C	// IN-BUFF MOV->LEFT
AND       M0191A	// T)ÅõÀÔ/¹èÃâ
OR LOAD
LOAD      M04022	// L_P&P Y PUT POS
OR        F00099
AND LOAD
OUT       P0009E	// OUT-BUFF MOV->LEFT (L-P&P)

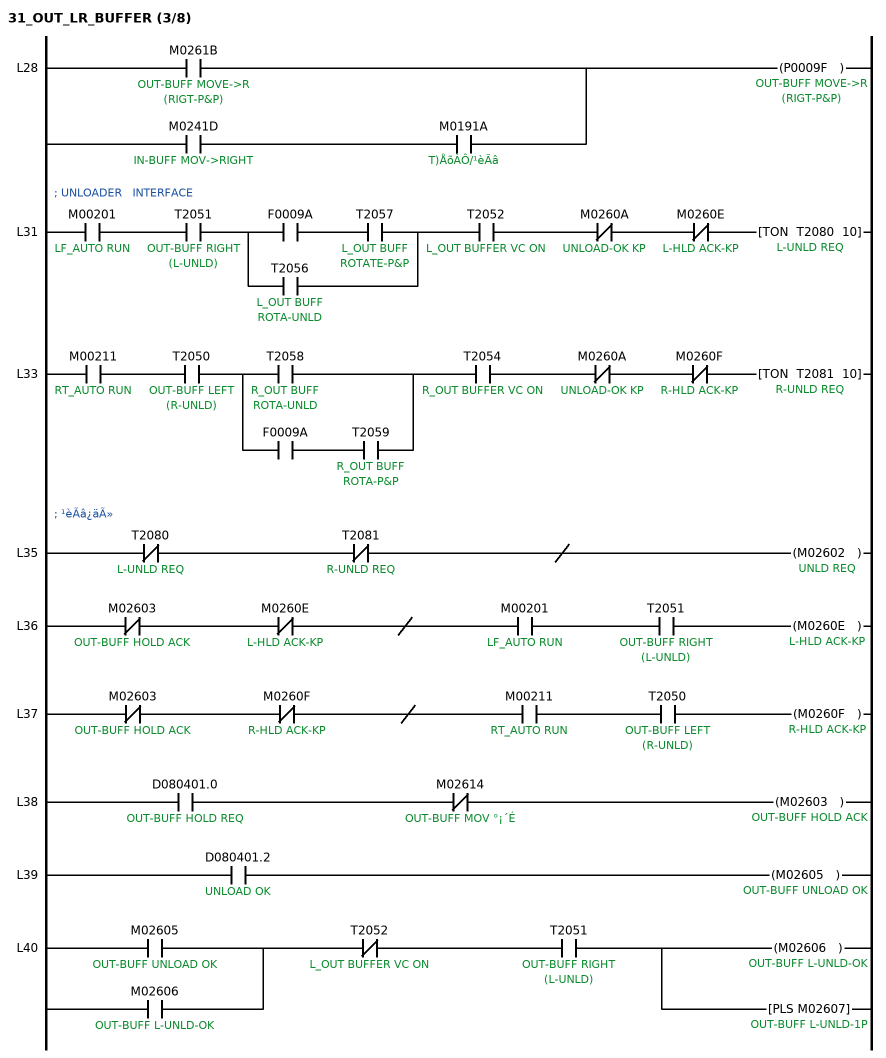
; L28
LOAD      M0261B	// OUT-BUFF MOVE->R (RIGT-P&P)
LOAD      M0241D	// IN-BUFF MOV->RIGHT
AND       M0191A	// T)ÅõÀÔ/¹èÃâ
OR LOAD
OUT       P0009F	// OUT-BUFF MOVE->R (RIGT-P&P)
//  UNLOADER   INTERFACE
; L31
LOAD      M00201	// LF_AUTO RUN
AND       T2051	// OUT-BUFF RIGHT (L-UNLD)
LOAD      F0009A
AND       T2057	// L_OUT BUFF ROTATE-P&P
OR        T2056	// L_OUT BUFF ROTA-UNLD
AND LOAD
AND       T2052	// L_OUT BUFFER VC ON
AND NOT   M0260A	// UNLOAD-OK KP
AND NOT   M0260E	// L-HLD ACK-KP
TON       T2080 10	// L-UNLD REQ
; L33
LOAD      M00211	// RT_AUTO RUN
AND       T2050	// OUT-BUFF LEFT (R-UNLD)
LOAD      T2058	// R_OUT BUFF ROTA-UNLD
LOAD      F0009A
AND       T2059	// R_OUT BUFF ROTA-P&P
OR LOAD
AND LOAD
AND       T2054	// R_OUT BUFFER VC ON
AND NOT   M0260A	// UNLOAD-OK KP
AND NOT   M0260F	// R-HLD ACK-KP
TON       T2081 10	// R-UNLD REQ
; L35
LOAD NOT  T2080	// L-UNLD REQ
AND NOT   T2081	// R-UNLD REQ
NOT
OUT       M02602	// UNLD REQ
// output comment: ¹èÃâ¿äÃ»
; L36
LOAD NOT  M02603	// OUT-BUFF HOLD ACK
AND NOT   M0260E	// L-HLD ACK-KP
NOT
AND       M00201	// LF_AUTO RUN
AND       T2051	// OUT-BUFF RIGHT (L-UNLD)
OUT       M0260E	// L-HLD ACK-KP
; L37
LOAD NOT  M02603	// OUT-BUFF HOLD ACK
AND NOT   M0260F	// R-HLD ACK-KP
NOT
AND       M00211	// RT_AUTO RUN
AND       T2050	// OUT-BUFF LEFT (R-UNLD)
OUT       M0260F	// R-HLD ACK-KP
; L38
LOAD      D080401.0	// OUT-BUFF HOLD REQ
AND NOT   M02614	// OUT-BUFF MOV °¡´É
OUT       M02603	// OUT-BUFF HOLD ACK
; L39
LOAD      D080401.2	// UNLOAD OK
OUT       M02605	// OUT-BUFF UNLOAD OK
; L40
LOAD      M02605	// OUT-BUFF UNLOAD OK
OR        M02606	// OUT-BUFF L-UNLD-OK
AND NOT   T2052	// L_OUT BUFFER VC ON
AND       T2051	// OUT-BUFF RIGHT (L-UNLD)
OUT       M02606	// OUT-BUFF L-UNLD-OK
OUTP      M02607	// OUT-BUFF L-UNLD-1P

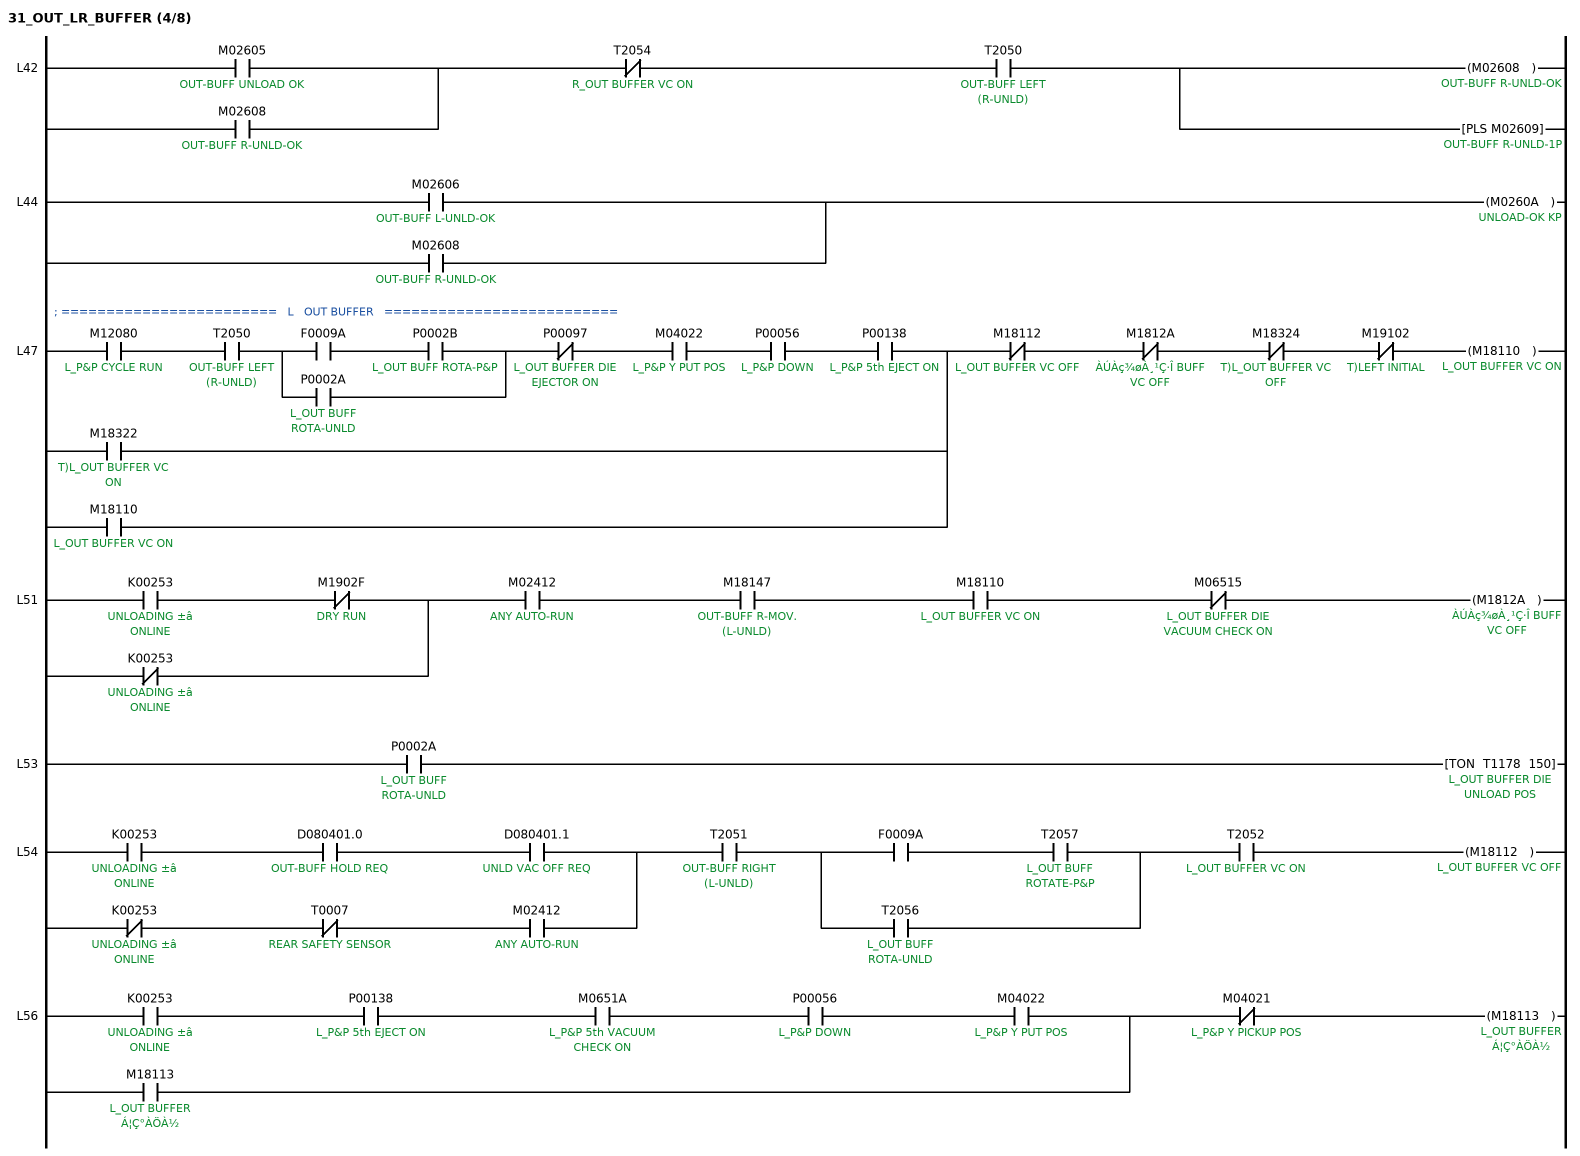
; L42
LOAD      M02605	// OUT-BUFF UNLOAD OK
OR        M02608	// OUT-BUFF R-UNLD-OK
AND NOT   T2054	// R_OUT BUFFER VC ON
AND       T2050	// OUT-BUFF LEFT (R-UNLD)
OUT       M02608	// OUT-BUFF R-UNLD-OK
OUTP      M02609	// OUT-BUFF R-UNLD-1P
; L44
LOAD      M02606	// OUT-BUFF L-UNLD-OK
OR        M02608	// OUT-BUFF R-UNLD-OK
OUT       M0260A	// UNLOAD-OK KP
// ========================   L   OUT BUFFER   ==========================
; L47
LOAD      M12080	// L_P&P CYCLE RUN
AND       T2050	// OUT-BUFF LEFT (R-UNLD)
LOAD      F0009A
AND       P0002B	// L_OUT BUFF ROTA-P&P
OR        P0002A	// L_OUT BUFF ROTA-UNLD
AND LOAD
AND NOT   P00097	// L_OUT BUFFER DIE EJECTOR ON
AND       M04022	// L_P&P Y PUT POS
AND       P00056	// L_P&P DOWN
AND       P00138	// L_P&P 5th EJECT ON
OR        M18322	// T)L_OUT BUFFER VC ON
OR        M18110	// L_OUT BUFFER VC ON
AND NOT   M18112	// L_OUT BUFFER VC OFF
AND NOT   M1812A	// ÀÚÀç¾øÀ¸¹Ç·Î BUFF VC OFF
AND NOT   M18324	// T)L_OUT BUFFER VC OFF
AND NOT   M19102	// T)LEFT INITIAL
OUT       M18110	// L_OUT BUFFER VC ON
; L51
LOAD      K00253	// UNLOADING ±â ONLINE
AND NOT   M1902F	// DRY RUN
OR NOT    K00253	// UNLOADING ±â ONLINE
AND       M02412	// ANY AUTO-RUN
AND       M18147	// OUT-BUFF R-MOV.  (L-UNLD)
AND       M18110	// L_OUT BUFFER VC ON
AND NOT   M06515	// L_OUT BUFFER DIE VACUUM CHECK ON
OUT       M1812A	// ÀÚÀç¾øÀ¸¹Ç·Î BUFF VC OFF
; L53
LOAD      P0002A	// L_OUT BUFF ROTA-UNLD
TON       T1178 150	// L_OUT BUFFER DIE UNLOAD POS
; L54
LOAD      K00253	// UNLOADING ±â ONLINE
AND       D080401.0	// OUT-BUFF HOLD REQ
AND       D080401.1	// UNLD VAC OFF REQ
LOAD NOT  K00253	// UNLOADING ±â ONLINE
AND NOT   T0007	// REAR SAFETY SENSOR
AND       M02412	// ANY AUTO-RUN
OR LOAD
AND       T2051	// OUT-BUFF RIGHT (L-UNLD)
LOAD      F0009A
AND       T2057	// L_OUT BUFF ROTATE-P&P
OR        T2056	// L_OUT BUFF ROTA-UNLD
AND LOAD
AND       T2052	// L_OUT BUFFER VC ON
OUT       M18112	// L_OUT BUFFER VC OFF
; L56
LOAD      K00253	// UNLOADING ±â ONLINE
AND       P00138	// L_P&P 5th EJECT ON
AND       M0651A	// L_P&P 5th VACUUM CHECK ON
AND       P00056	// L_P&P DOWN
AND       M04022	// L_P&P Y PUT POS
OR        M18113	// L_OUT BUFFER Á¦Ç°ÀÖÀ½
AND NOT   M04021	// L_P&P Y PICKUP POS
OUT       M18113	// L_OUT BUFFER Á¦Ç°ÀÖÀ½

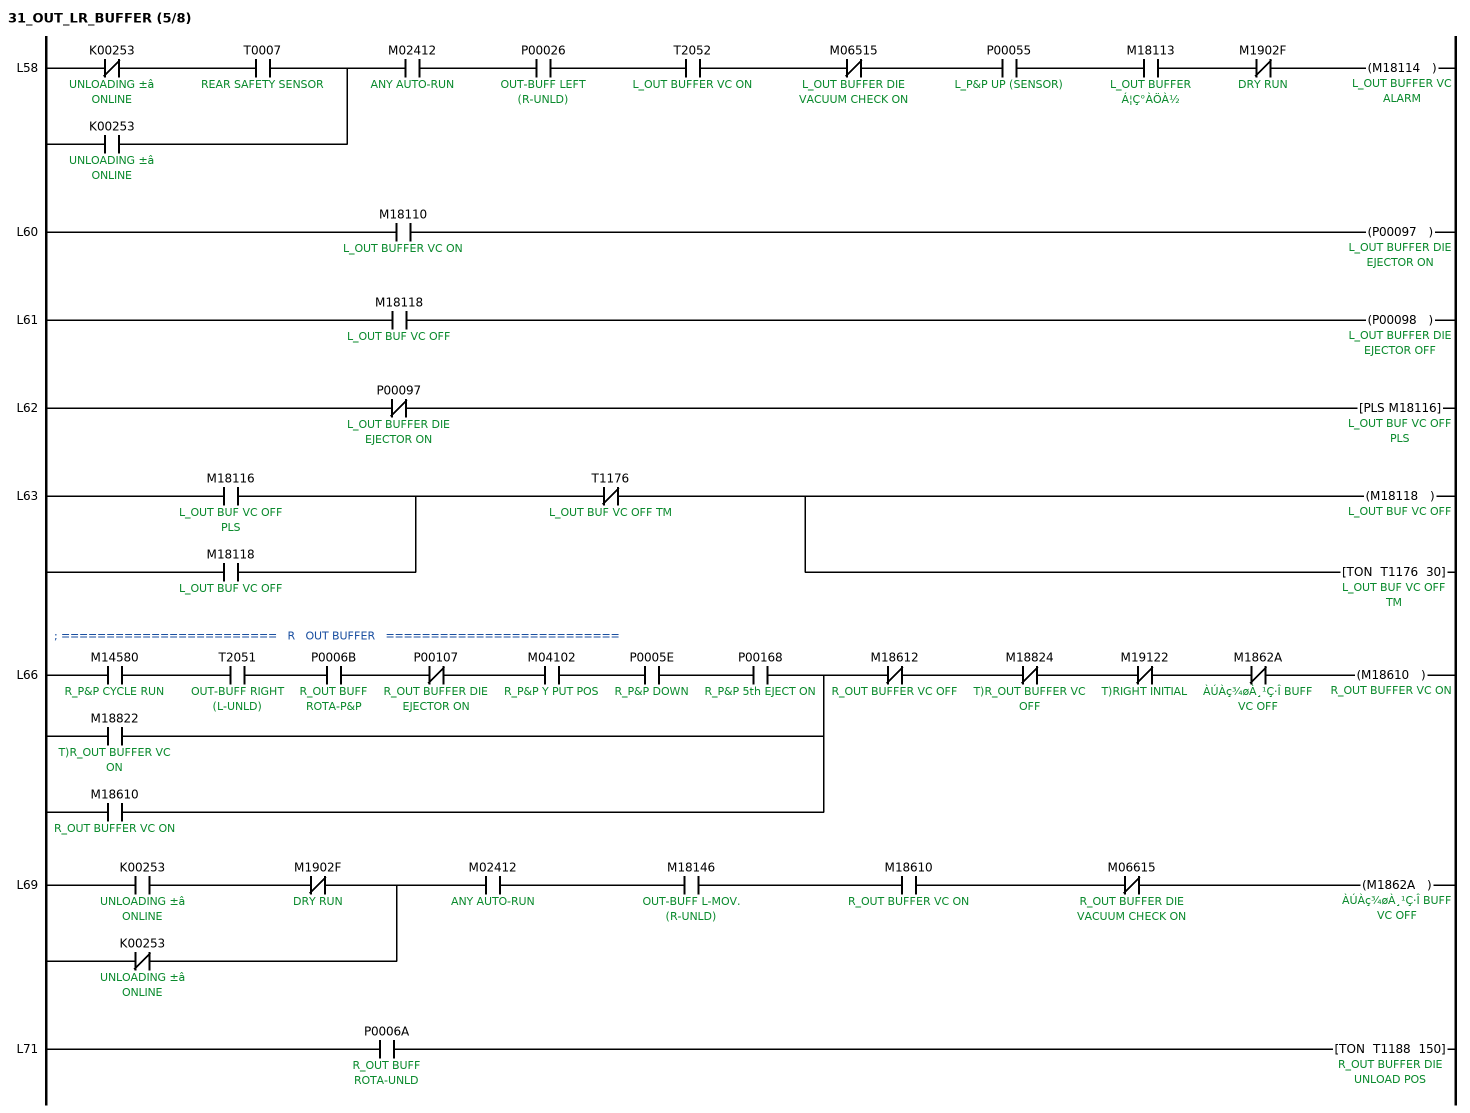
; L58
LOAD NOT  K00253	// UNLOADING ±â ONLINE
AND       T0007	// REAR SAFETY SENSOR
OR        K00253	// UNLOADING ±â ONLINE
AND       M02412	// ANY AUTO-RUN
AND       P00026	// OUT-BUFF LEFT (R-UNLD)
AND       T2052	// L_OUT BUFFER VC ON
AND NOT   M06515	// L_OUT BUFFER DIE VACUUM CHECK ON
AND       P00055	// L_P&P UP (SENSOR)
AND       M18113	// L_OUT BUFFER Á¦Ç°ÀÖÀ½
AND NOT   M1902F	// DRY RUN
OUT       M18114	// L_OUT BUFFER VC ALARM
; L60
LOAD      M18110	// L_OUT BUFFER VC ON
OUT       P00097	// L_OUT BUFFER DIE EJECTOR ON
; L61
LOAD      M18118	// L_OUT BUF VC OFF
OUT       P00098	// L_OUT BUFFER DIE EJECTOR OFF
; L62
LOAD NOT  P00097	// L_OUT BUFFER DIE EJECTOR ON
OUTP      M18116	// L_OUT BUF VC OFF PLS
; L63
LOAD      M18116	// L_OUT BUF VC OFF PLS
OR        M18118	// L_OUT BUF VC OFF
AND NOT   T1176	// L_OUT BUF VC OFF TM
OUT       M18118	// L_OUT BUF VC OFF
TON       T1176 30	// L_OUT BUF VC OFF TM
// ========================   R   OUT BUFFER   ==========================
; L66
LOAD      M14580	// R_P&P CYCLE RUN
AND       T2051	// OUT-BUFF RIGHT (L-UNLD)
AND       P0006B	// R_OUT BUFF ROTA-P&P
AND NOT   P00107	// R_OUT BUFFER DIE EJECTOR ON
AND       M04102	// R_P&P Y PUT POS
AND       P0005E	// R_P&P DOWN
AND       P00168	// R_P&P 5th EJECT ON
OR        M18822	// T)R_OUT BUFFER VC ON
OR        M18610	// R_OUT BUFFER VC ON
AND NOT   M18612	// R_OUT BUFFER VC OFF
AND NOT   M18824	// T)R_OUT BUFFER VC OFF
AND NOT   M19122	// T)RIGHT INITIAL
AND NOT   M1862A	// ÀÚÀç¾øÀ¸¹Ç·Î BUFF VC OFF
OUT       M18610	// R_OUT BUFFER VC ON
; L69
LOAD      K00253	// UNLOADING ±â ONLINE
AND NOT   M1902F	// DRY RUN
OR NOT    K00253	// UNLOADING ±â ONLINE
AND       M02412	// ANY AUTO-RUN
AND       M18146	// OUT-BUFF L-MOV. (R-UNLD)
AND       M18610	// R_OUT BUFFER VC ON
AND NOT   M06615	// R_OUT BUFFER DIE VACUUM CHECK ON
OUT       M1862A	// ÀÚÀç¾øÀ¸¹Ç·Î BUFF VC OFF
; L71
LOAD      P0006A	// R_OUT BUFF ROTA-UNLD
TON       T1188 150	// R_OUT BUFFER DIE UNLOAD POS

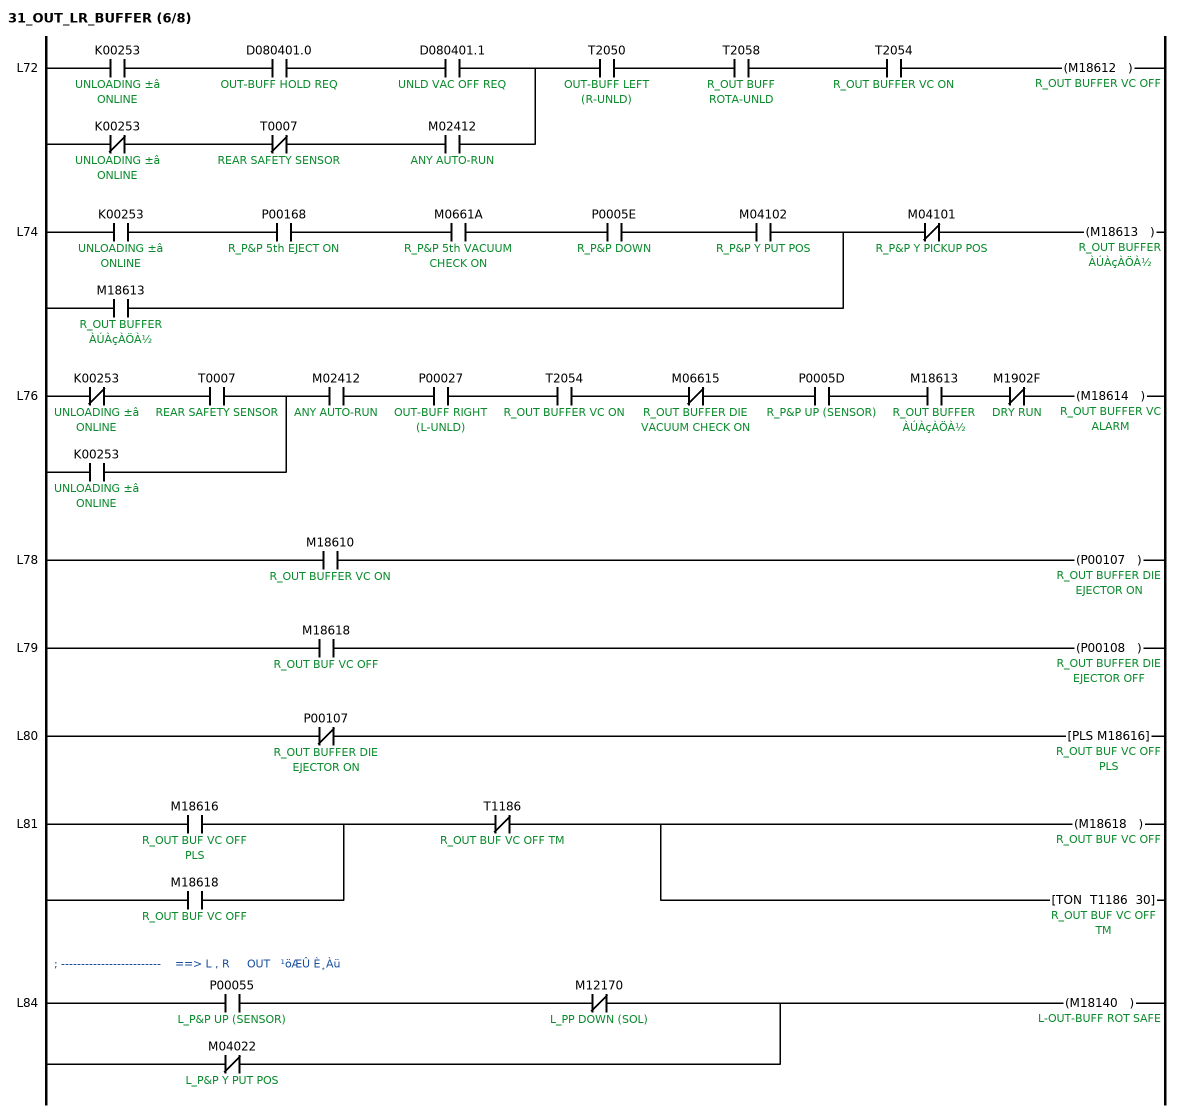
; L72
LOAD      K00253	// UNLOADING ±â ONLINE
AND       D080401.0	// OUT-BUFF HOLD REQ
AND       D080401.1	// UNLD VAC OFF REQ
LOAD NOT  K00253	// UNLOADING ±â ONLINE
AND NOT   T0007	// REAR SAFETY SENSOR
AND       M02412	// ANY AUTO-RUN
OR LOAD
AND       T2050	// OUT-BUFF LEFT (R-UNLD)
AND       T2058	// R_OUT BUFF ROTA-UNLD
AND       T2054	// R_OUT BUFFER VC ON
OUT       M18612	// R_OUT BUFFER VC OFF
; L74
LOAD      K00253	// UNLOADING ±â ONLINE
AND       P00168	// R_P&P 5th EJECT ON
AND       M0661A	// R_P&P 5th VACUUM CHECK ON
AND       P0005E	// R_P&P DOWN
AND       M04102	// R_P&P Y PUT POS
OR        M18613	// R_OUT BUFFER ÀÚÀçÀÖÀ½
AND NOT   M04101	// R_P&P Y PICKUP POS
OUT       M18613	// R_OUT BUFFER ÀÚÀçÀÖÀ½
; L76
LOAD NOT  K00253	// UNLOADING ±â ONLINE
AND       T0007	// REAR SAFETY SENSOR
OR        K00253	// UNLOADING ±â ONLINE
AND       M02412	// ANY AUTO-RUN
AND       P00027	// OUT-BUFF RIGHT (L-UNLD)
AND       T2054	// R_OUT BUFFER VC ON
AND NOT   M06615	// R_OUT BUFFER DIE VACUUM CHECK ON
AND       P0005D	// R_P&P UP (SENSOR)
AND       M18613	// R_OUT BUFFER ÀÚÀçÀÖÀ½
AND NOT   M1902F	// DRY RUN
OUT       M18614	// R_OUT BUFFER VC ALARM
; L78
LOAD      M18610	// R_OUT BUFFER VC ON
OUT       P00107	// R_OUT BUFFER DIE EJECTOR ON
; L79
LOAD      M18618	// R_OUT BUF VC OFF
OUT       P00108	// R_OUT BUFFER DIE EJECTOR OFF
; L80
LOAD NOT  P00107	// R_OUT BUFFER DIE EJECTOR ON
OUTP      M18616	// R_OUT BUF VC OFF PLS
; L81
LOAD      M18616	// R_OUT BUF VC OFF PLS
OR        M18618	// R_OUT BUF VC OFF
AND NOT   T1186	// R_OUT BUF VC OFF TM
OUT       M18618	// R_OUT BUF VC OFF
TON       T1186 30	// R_OUT BUF VC OFF TM
// -------------------------    ==> L , R     OUT   ¹öÆÛ È¸Àü
; L84
LOAD      P00055	// L_P&P UP (SENSOR)
AND NOT   M12170	// L_PP DOWN (SOL)
OR NOT    M04022	// L_P&P Y PUT POS
OUT       M18140	// L-OUT-BUFF ROT SAFE

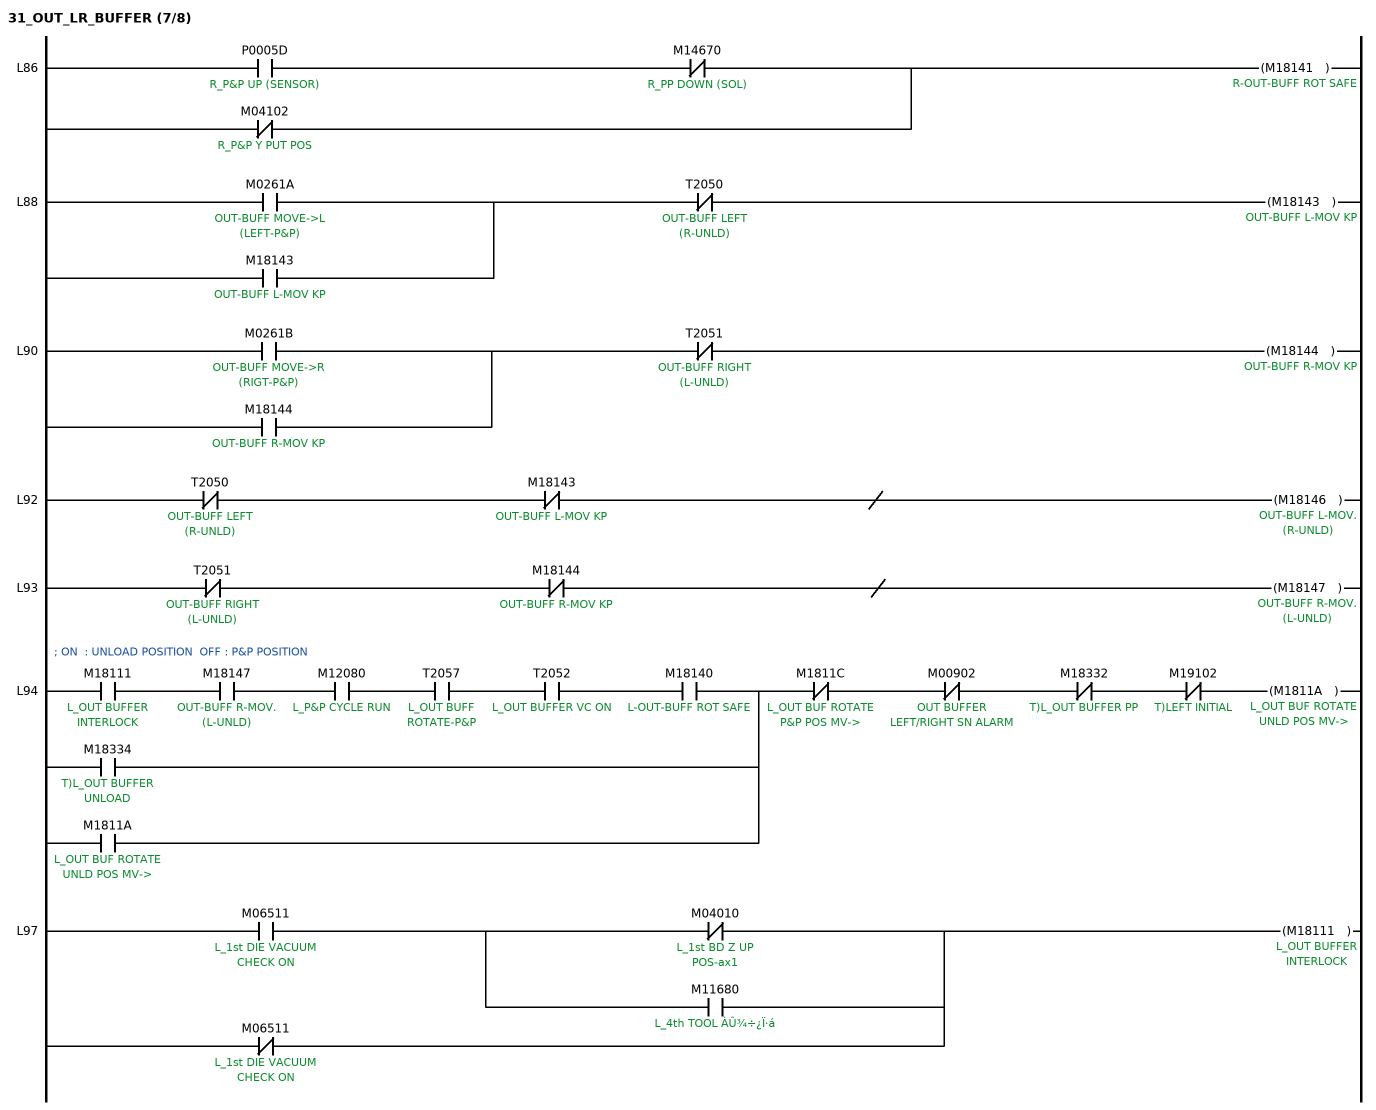
; L86
LOAD      P0005D	// R_P&P UP (SENSOR)
AND NOT   M14670	// R_PP DOWN (SOL)
OR NOT    M04102	// R_P&P Y PUT POS
OUT       M18141	// R-OUT-BUFF ROT SAFE
; L88
LOAD      M0261A	// OUT-BUFF MOVE->L (LEFT-P&P)
OR        M18143	// OUT-BUFF L-MOV KP
AND NOT   T2050	// OUT-BUFF LEFT (R-UNLD)
OUT       M18143	// OUT-BUFF L-MOV KP
; L90
LOAD      M0261B	// OUT-BUFF MOVE->R (RIGT-P&P)
OR        M18144	// OUT-BUFF R-MOV KP
AND NOT   T2051	// OUT-BUFF RIGHT (L-UNLD)
OUT       M18144	// OUT-BUFF R-MOV KP
; L92
LOAD NOT  T2050	// OUT-BUFF LEFT (R-UNLD)
AND NOT   M18143	// OUT-BUFF L-MOV KP
NOT
OUT       M18146	// OUT-BUFF L-MOV. (R-UNLD)
; L93
LOAD NOT  T2051	// OUT-BUFF RIGHT (L-UNLD)
AND NOT   M18144	// OUT-BUFF R-MOV KP
NOT
OUT       M18147	// OUT-BUFF R-MOV.  (L-UNLD)
; L94
LOAD      M18111	// L_OUT BUFFER INTERLOCK
AND       M18147	// OUT-BUFF R-MOV.  (L-UNLD)
AND       M12080	// L_P&P CYCLE RUN
AND       T2057	// L_OUT BUFF ROTATE-P&P
AND       T2052	// L_OUT BUFFER VC ON
AND       M18140	// L-OUT-BUFF ROT SAFE
OR        M18334	// T)L_OUT BUFFER UNLOAD
OR        M1811A	// L_OUT BUF ROTATE UNLD POS MV->
AND NOT   M1811C	// L_OUT BUF ROTATE P&P POS MV->
AND NOT   M00902	// OUT BUFFER LEFT/RIGHT SN ALARM
AND NOT   M18332	// T)L_OUT BUFFER PP
AND NOT   M19102	// T)LEFT INITIAL
OUT       M1811A	// L_OUT BUF ROTATE UNLD POS MV->
// output comment: ON  : UNLOAD POSITION  OFF : P&P POSITION
; L97
LOAD      M06511	// L_1st DIE VACUUM CHECK ON
LOAD NOT  M04010	// L_1st BD Z UP POS-ax1
OR        M11680	// L_4th TOOL ÀÛ¾÷¿Ï·á
AND LOAD
OR NOT    M06511	// L_1st DIE VACUUM CHECK ON
OUT       M18111	// L_OUT BUFFER INTERLOCK

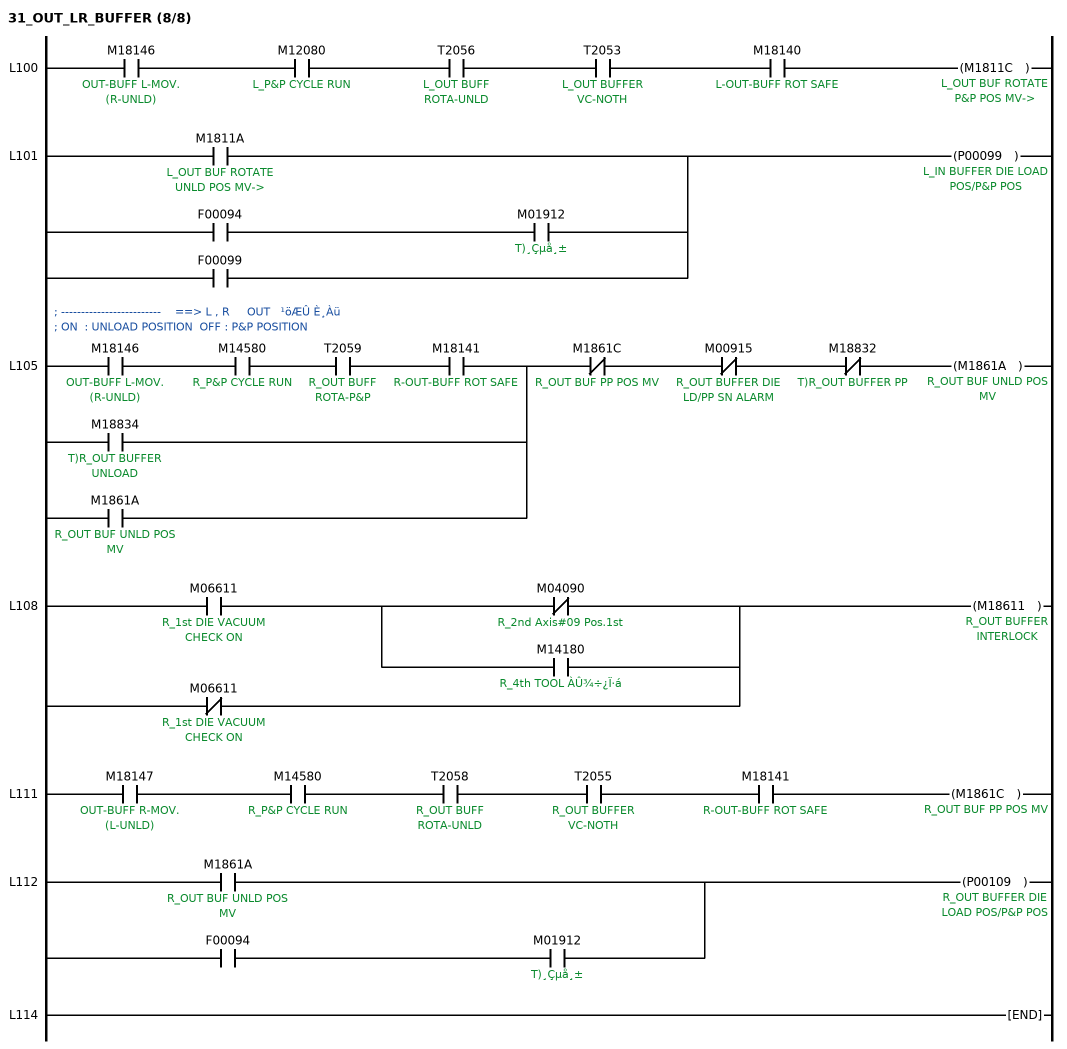
; L100
LOAD      M18146	// OUT-BUFF L-MOV. (R-UNLD)
AND       M12080	// L_P&P CYCLE RUN
AND       T2056	// L_OUT BUFF ROTA-UNLD
AND       T2053	// L_OUT BUFFER VC-NOTH
AND       M18140	// L-OUT-BUFF ROT SAFE
OUT       M1811C	// L_OUT BUF ROTATE P&P POS MV->
; L101
LOAD      M1811A	// L_OUT BUF ROTATE UNLD POS MV->
LOAD      F00094
AND       M01912	// T)¸Çµå¸±
OR LOAD
OR        F00099
OUT       P00099	// L_IN BUFFER DIE LOAD POS/P&P POS
// -------------------------    ==> L , R     OUT   ¹öÆÛ È¸Àü
; L105
LOAD      M18146	// OUT-BUFF L-MOV. (R-UNLD)
AND       M14580	// R_P&P CYCLE RUN
AND       T2059	// R_OUT BUFF ROTA-P&P
AND       M18141	// R-OUT-BUFF ROT SAFE
OR        M18834	// T)R_OUT BUFFER UNLOAD
OR        M1861A	// R_OUT BUF UNLD POS MV
AND NOT   M1861C	// R_OUT BUF PP POS MV
AND NOT   M00915	// R_OUT BUFFER DIE LD/PP SN ALARM
AND NOT   M18832	// T)R_OUT BUFFER PP
OUT       M1861A	// R_OUT BUF UNLD POS MV
// output comment: ON  : UNLOAD POSITION  OFF : P&P POSITION
; L108
LOAD      M06611	// R_1st DIE VACUUM CHECK ON
LOAD NOT  M04090	// R_2nd Axis#09 Pos.1st
OR        M14180	// R_4th TOOL ÀÛ¾÷¿Ï·á
AND LOAD
OR NOT    M06611	// R_1st DIE VACUUM CHECK ON
OUT       M18611	// R_OUT BUFFER INTERLOCK
; L111
LOAD      M18147	// OUT-BUFF R-MOV.  (L-UNLD)
AND       M14580	// R_P&P CYCLE RUN
AND       T2058	// R_OUT BUFF ROTA-UNLD
AND       T2055	// R_OUT BUFFER VC-NOTH
AND       M18141	// R-OUT-BUFF ROT SAFE
OUT       M1861C	// R_OUT BUF PP POS MV
; L112
LOAD      M1861A	// R_OUT BUF UNLD POS MV
LOAD      F00094
AND       M01912	// T)¸Çµå¸±
OR LOAD
OUT       P00109	// R_OUT BUFFER DIE LOAD POS/P&P POS
; L114
END

PROGRAM 40_2D_CODE (task: ½ºÄµ ÇÁ·Î±×·¥)

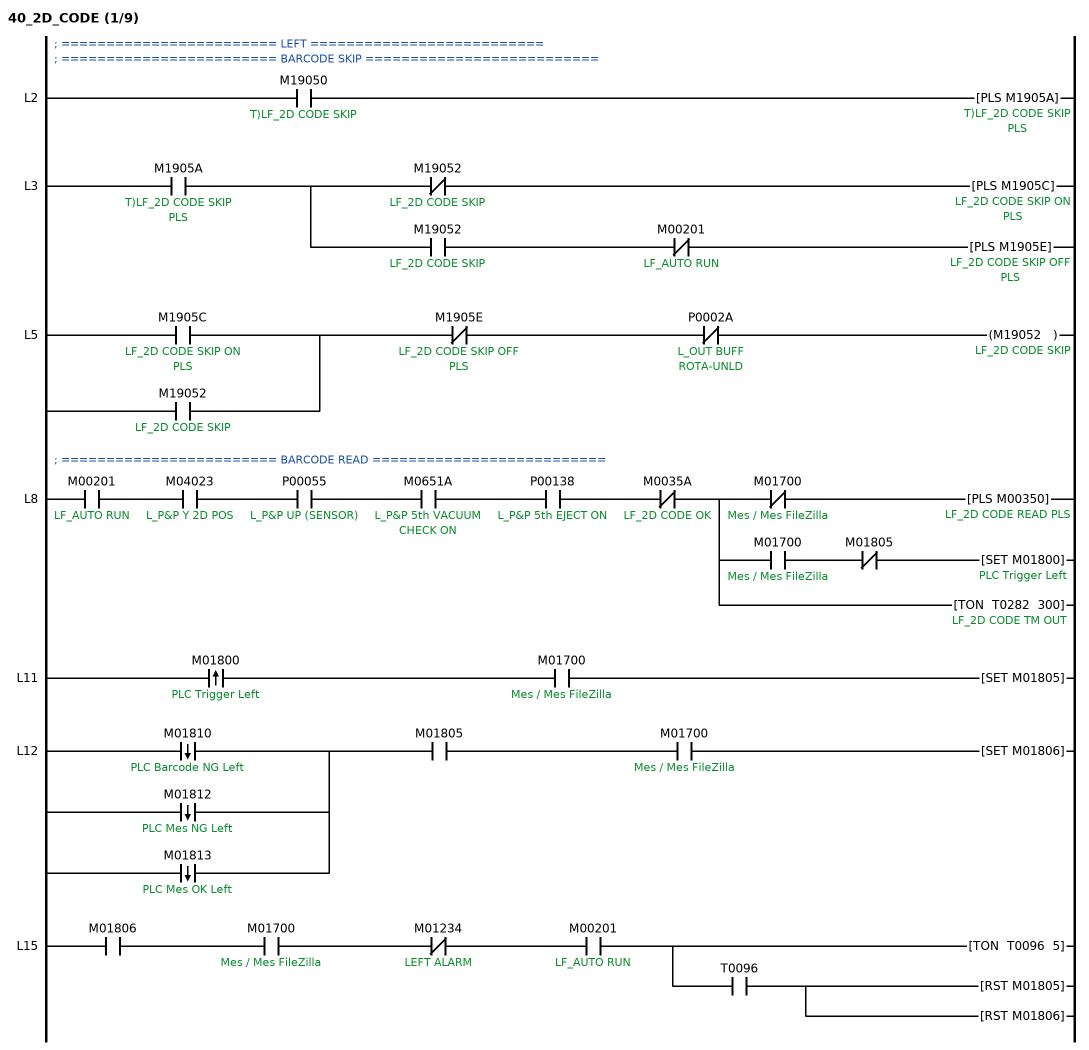
// ======================== LEFT ==========================
// ======================== BARCODE SKIP ==========================
; L2
LOAD      M19050	// T)LF_2D CODE SKIP
OUTP      M1905A	// T)LF_2D CODE SKIP PLS
; L3
LOAD      M1905A	// T)LF_2D CODE SKIP PLS
MPUSH
AND NOT   M19052	// LF_2D CODE SKIP
OUTP      M1905C	// LF_2D CODE SKIP ON PLS
MPOP
AND       M19052	// LF_2D CODE SKIP
AND NOT   M00201	// LF_AUTO RUN
OUTP      M1905E	// LF_2D CODE SKIP OFF PLS
; L5
LOAD      M1905C	// LF_2D CODE SKIP ON PLS
OR        M19052	// LF_2D CODE SKIP
AND NOT   M1905E	// LF_2D CODE SKIP OFF PLS
AND NOT   P0002A	// L_OUT BUFF ROTA-UNLD
OUT       M19052	// LF_2D CODE SKIP
// ======================== BARCODE READ ==========================
; L8
LOAD      M00201	// LF_AUTO RUN
AND       M04023	// L_P&P Y 2D POS
AND       P00055	// L_P&P UP (SENSOR)
AND       M0651A	// L_P&P 5th VACUUM CHECK ON
AND       P00138	// L_P&P 5th EJECT ON
AND NOT   M0035A	// LF_2D CODE OK
MPUSH
AND NOT   M01700	// Mes / Mes FileZilla
OUTP      M00350	// LF_2D CODE READ PLS
MLOAD
AND       M01700	// Mes / Mes FileZilla
AND NOT   M01805
SET       M01800	// PLC Trigger Left
MPOP
TON       T0282 300	// LF_2D CODE TM OUT
; L11
LOADP     M01800	// PLC Trigger Left
AND       M01700	// Mes / Mes FileZilla
SET       M01805
; L12
LOADN     M01810	// PLC Barcode NG Left
ORN       M01812	// PLC Mes NG Left
ORN       M01813	// PLC Mes OK Left
AND       M01805
AND       M01700	// Mes / Mes FileZilla
SET       M01806
; L15
LOAD      M01806
AND       M01700	// Mes / Mes FileZilla
AND NOT   M01234	// LEFT ALARM
AND       M00201	// LF_AUTO RUN
TON       T0096 5
AND       T0096
RST       M01805
RST       M01806

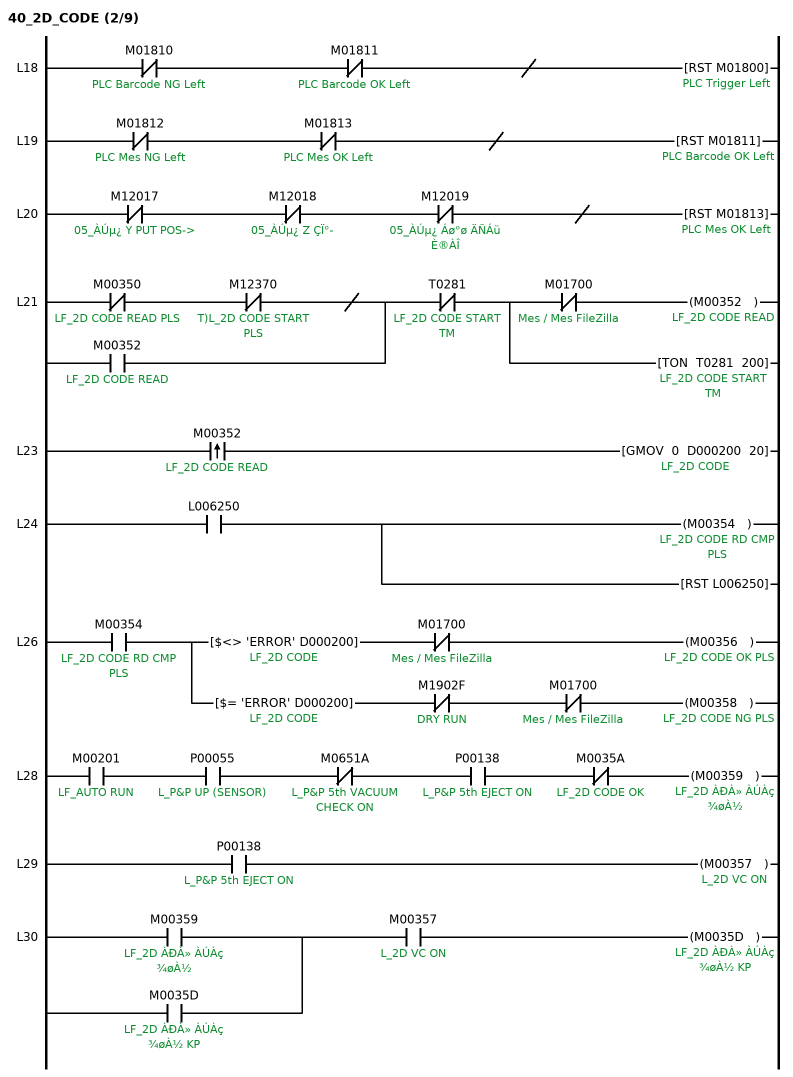
; L18
LOAD NOT  M01810	// PLC Barcode NG Left
AND NOT   M01811	// PLC Barcode OK Left
NOT
RST       M01800	// PLC Trigger Left
; L19
LOAD NOT  M01812	// PLC Mes NG Left
AND NOT   M01813	// PLC Mes OK Left
NOT
RST       M01811	// PLC Barcode OK Left
; L20
LOAD NOT  M12017	// 05_ÀÚµ¿ Y PUT POS->
AND NOT   M12018	// 05_ÀÚµ¿ Z ÇÏ°­
AND NOT   M12019	// 05_ÀÚµ¿ Áø°ø ÄÑÁü È®ÀÎ
NOT
RST       M01813	// PLC Mes OK Left
; L21
LOAD NOT  M00350	// LF_2D CODE READ PLS
AND NOT   M12370	// T)L_2D CODE START PLS
NOT
OR        M00352	// LF_2D CODE READ
AND NOT   T0281	// LF_2D CODE START TM
MPUSH
AND NOT   M01700	// Mes / Mes FileZilla
OUT       M00352	// LF_2D CODE READ
MPOP
TON       T0281 200	// LF_2D CODE START TM
; L23
LOADP     M00352	// LF_2D CODE READ
GMOV      0 D000200 20	// LF_2D CODE
; L24
LOAD      L006250
OUT       M00354	// LF_2D CODE RD CMP PLS
RST       L006250
; L26
LOAD      M00354	// LF_2D CODE RD CMP PLS
MPUSH
AND$<>    'ERROR' D000200	// LF_2D CODE
AND NOT   M01700	// Mes / Mes FileZilla
OUT       M00356	// LF_2D CODE OK PLS
MPOP
AND$=     'ERROR' D000200	// LF_2D CODE
AND NOT   M1902F	// DRY RUN
AND NOT   M01700	// Mes / Mes FileZilla
OUT       M00358	// LF_2D CODE NG PLS
; L28
LOAD      M00201	// LF_AUTO RUN
AND       P00055	// L_P&P UP (SENSOR)
AND NOT   M0651A	// L_P&P 5th VACUUM CHECK ON
AND       P00138	// L_P&P 5th EJECT ON
AND NOT   M0035A	// LF_2D CODE OK
OUT       M00359	// LF_2D ÀÐÀ» ÀÚÀç ¾øÀ½
; L29
LOAD      P00138	// L_P&P 5th EJECT ON
OUT       M00357	// L_2D VC ON
; L30
LOAD      M00359	// LF_2D ÀÐÀ» ÀÚÀç ¾øÀ½
OR        M0035D	// LF_2D ÀÐÀ» ÀÚÀç ¾øÀ½ KP
AND       M00357	// L_2D VC ON
OUT       M0035D	// LF_2D ÀÐÀ» ÀÚÀç ¾øÀ½ KP

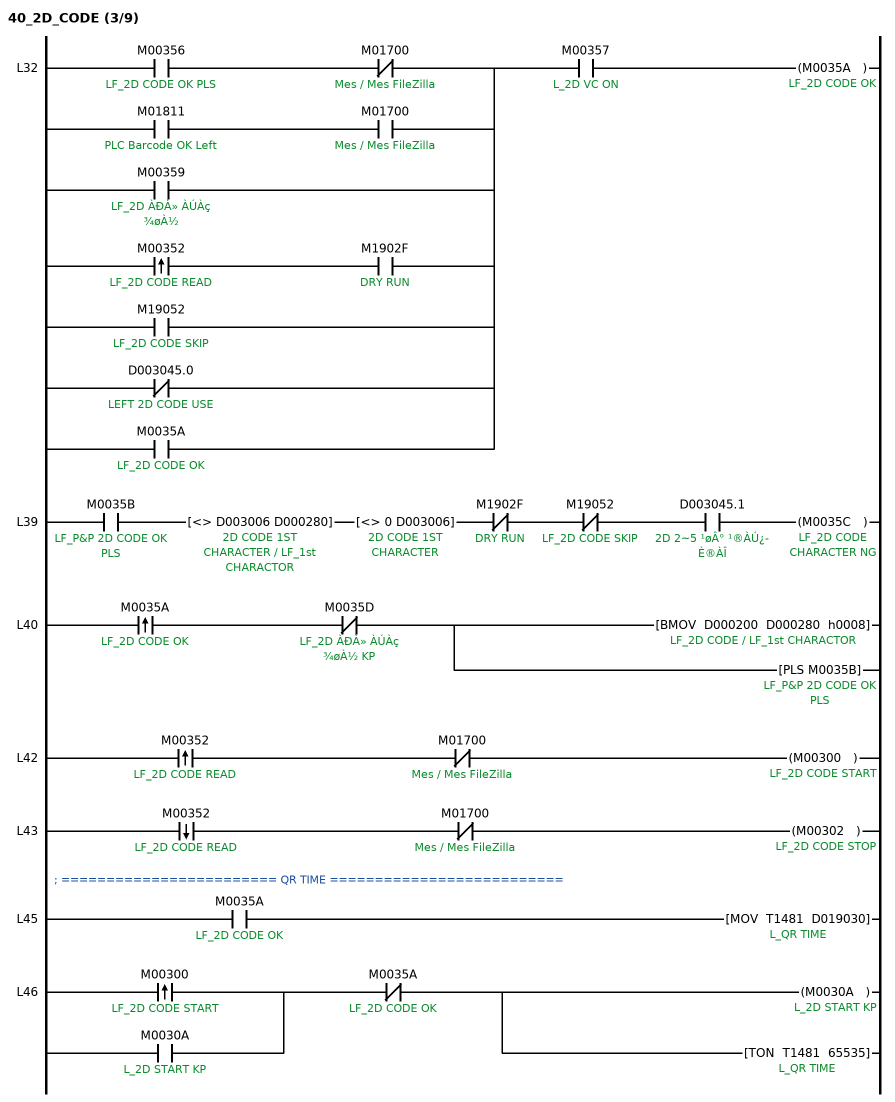
; L32
LOAD      M00356	// LF_2D CODE OK PLS
AND NOT   M01700	// Mes / Mes FileZilla
LOAD      M01811	// PLC Barcode OK Left
AND       M01700	// Mes / Mes FileZilla
OR LOAD
OR        M00359	// LF_2D ÀÐÀ» ÀÚÀç ¾øÀ½
LOADP     M00352	// LF_2D CODE READ
AND       M1902F	// DRY RUN
OR LOAD
OR        M19052	// LF_2D CODE SKIP
OR NOT    D003045.0	// LEFT 2D CODE USE
OR        M0035A	// LF_2D CODE OK
AND       M00357	// L_2D VC ON
OUT       M0035A	// LF_2D CODE OK
; L39
LOAD      M0035B	// LF_P&P 2D CODE OK PLS
AND<>     D003006 D000280	// 2D CODE 1ST CHARACTER / LF_1st CHARACTOR
AND<>     0 D003006	// 2D CODE 1ST CHARACTER
AND NOT   M1902F	// DRY RUN
AND NOT   M19052	// LF_2D CODE SKIP
AND       D003045.1	// 2D 2~5 ¹øÂ° ¹®ÀÚ¿­ È®ÀÎ
OUT       M0035C	// LF_2D CODE CHARACTER NG
; L40
LOADP     M0035A	// LF_2D CODE OK
AND NOT   M0035D	// LF_2D ÀÐÀ» ÀÚÀç ¾øÀ½ KP
BMOV      D000200 D000280 h0008	// LF_2D CODE / LF_1st CHARACTOR
OUTP      M0035B	// LF_P&P 2D CODE OK PLS
; L42
LOADP     M00352	// LF_2D CODE READ
AND NOT   M01700	// Mes / Mes FileZilla
OUT       M00300	// LF_2D CODE START
; L43
LOADN     M00352	// LF_2D CODE READ
AND NOT   M01700	// Mes / Mes FileZilla
OUT       M00302	// LF_2D CODE STOP
// ======================== QR TIME ==========================
; L45
LOAD      M0035A	// LF_2D CODE OK
MOV       T1481 D019030	// L_QR TIME
; L46
LOADP     M00300	// LF_2D CODE START
OR        M0030A	// L_2D START KP
AND NOT   M0035A	// LF_2D CODE OK
OUT       M0030A	// L_2D START KP
TON       T1481 65535	// L_QR TIME

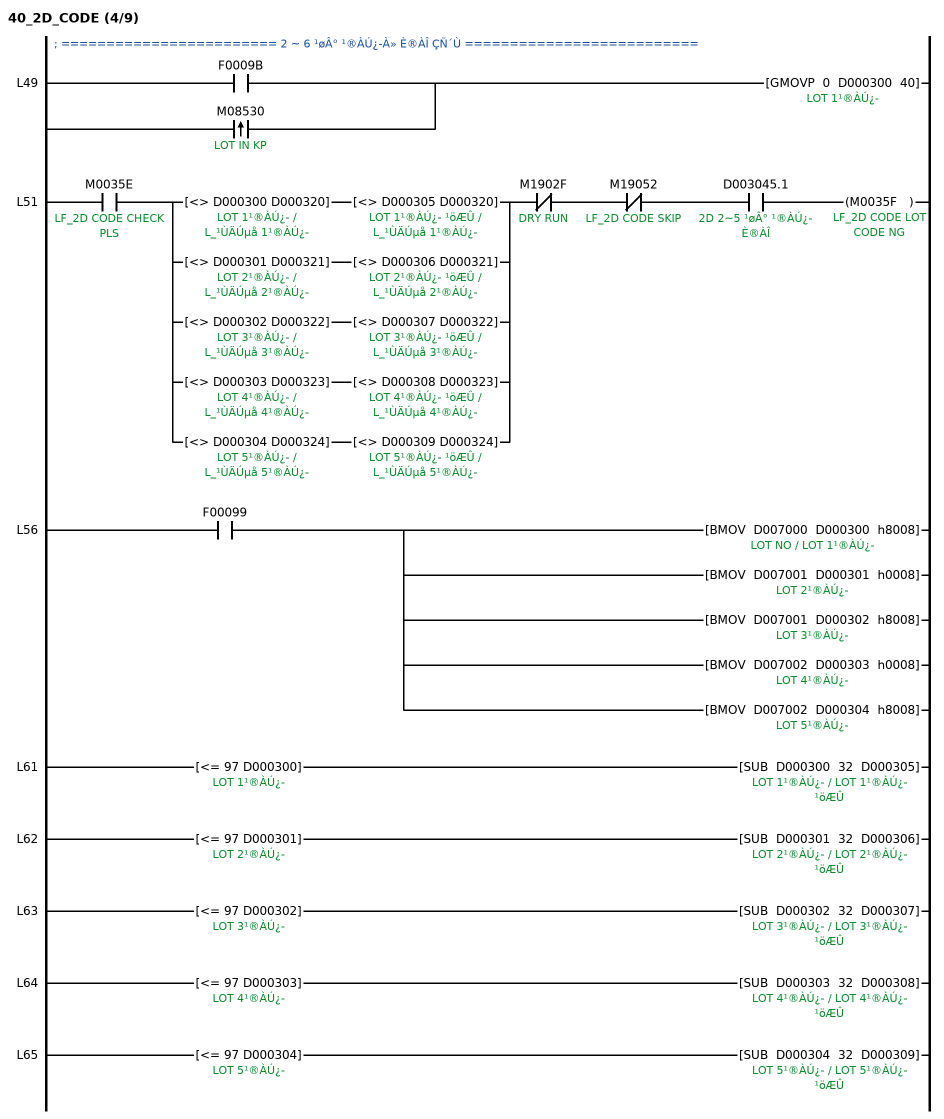
// ======================== 2 ~ 6 ¹øÂ° ¹®ÀÚ¿­À» È®ÀÎ ÇÑ´Ù ==========================
; L49
LOAD      F0009B
ORP       M08530	// LOT IN KP
GMOVP     0 D000300 40	// LOT 1¹®ÀÚ¿­
; L51
LOAD      M0035E	// LF_2D CODE CHECK PLS
LOAD<>    D000300 D000320	// LOT 1¹®ÀÚ¿­ / L_¹ÙÄÚµå 1¹®ÀÚ¿­
AND<>     D000305 D000320	// LOT 1¹®ÀÚ¿­ ¹öÆÛ / L_¹ÙÄÚµå 1¹®ÀÚ¿­
LOAD<>    D000301 D000321	// LOT 2¹®ÀÚ¿­ / L_¹ÙÄÚµå 2¹®ÀÚ¿­
AND<>     D000306 D000321	// LOT 2¹®ÀÚ¿­ ¹öÆÛ / L_¹ÙÄÚµå 2¹®ÀÚ¿­
OR LOAD
LOAD<>    D000302 D000322	// LOT 3¹®ÀÚ¿­ / L_¹ÙÄÚµå 3¹®ÀÚ¿­
AND<>     D000307 D000322	// LOT 3¹®ÀÚ¿­ ¹öÆÛ / L_¹ÙÄÚµå 3¹®ÀÚ¿­
OR LOAD
LOAD<>    D000303 D000323	// LOT 4¹®ÀÚ¿­ / L_¹ÙÄÚµå 4¹®ÀÚ¿­
AND<>     D000308 D000323	// LOT 4¹®ÀÚ¿­ ¹öÆÛ / L_¹ÙÄÚµå 4¹®ÀÚ¿­
OR LOAD
LOAD<>    D000304 D000324	// LOT 5¹®ÀÚ¿­ / L_¹ÙÄÚµå 5¹®ÀÚ¿­
AND<>     D000309 D000324	// LOT 5¹®ÀÚ¿­ ¹öÆÛ / L_¹ÙÄÚµå 5¹®ÀÚ¿­
OR LOAD
AND LOAD
AND NOT   M1902F	// DRY RUN
AND NOT   M19052	// LF_2D CODE SKIP
AND       D003045.1	// 2D 2~5 ¹øÂ° ¹®ÀÚ¿­ È®ÀÎ
OUT       M0035F	// LF_2D CODE LOT CODE NG
; L56
LOAD      F00099
BMOV      D007000 D000300 h8008	// LOT NO / LOT 1¹®ÀÚ¿­
BMOV      D007001 D000301 h0008	// LOT 2¹®ÀÚ¿­
BMOV      D007001 D000302 h8008	// LOT 3¹®ÀÚ¿­
BMOV      D007002 D000303 h0008	// LOT 4¹®ÀÚ¿­
BMOV      D007002 D000304 h8008	// LOT 5¹®ÀÚ¿­
; L61
LOAD<=    97 D000300	// LOT 1¹®ÀÚ¿­
SUB       D000300 32 D000305	// LOT 1¹®ÀÚ¿­ / LOT 1¹®ÀÚ¿­ ¹öÆÛ
; L62
LOAD<=    97 D000301	// LOT 2¹®ÀÚ¿­
SUB       D000301 32 D000306	// LOT 2¹®ÀÚ¿­ / LOT 2¹®ÀÚ¿­ ¹öÆÛ
; L63
LOAD<=    97 D000302	// LOT 3¹®ÀÚ¿­
SUB       D000302 32 D000307	// LOT 3¹®ÀÚ¿­ / LOT 3¹®ÀÚ¿­ ¹öÆÛ
; L64
LOAD<=    97 D000303	// LOT 4¹®ÀÚ¿­
SUB       D000303 32 D000308	// LOT 4¹®ÀÚ¿­ / LOT 4¹®ÀÚ¿­ ¹öÆÛ
; L65
LOAD<=    97 D000304	// LOT 5¹®ÀÚ¿­
SUB       D000304 32 D000309	// LOT 5¹®ÀÚ¿­ / LOT 5¹®ÀÚ¿­ ¹öÆÛ

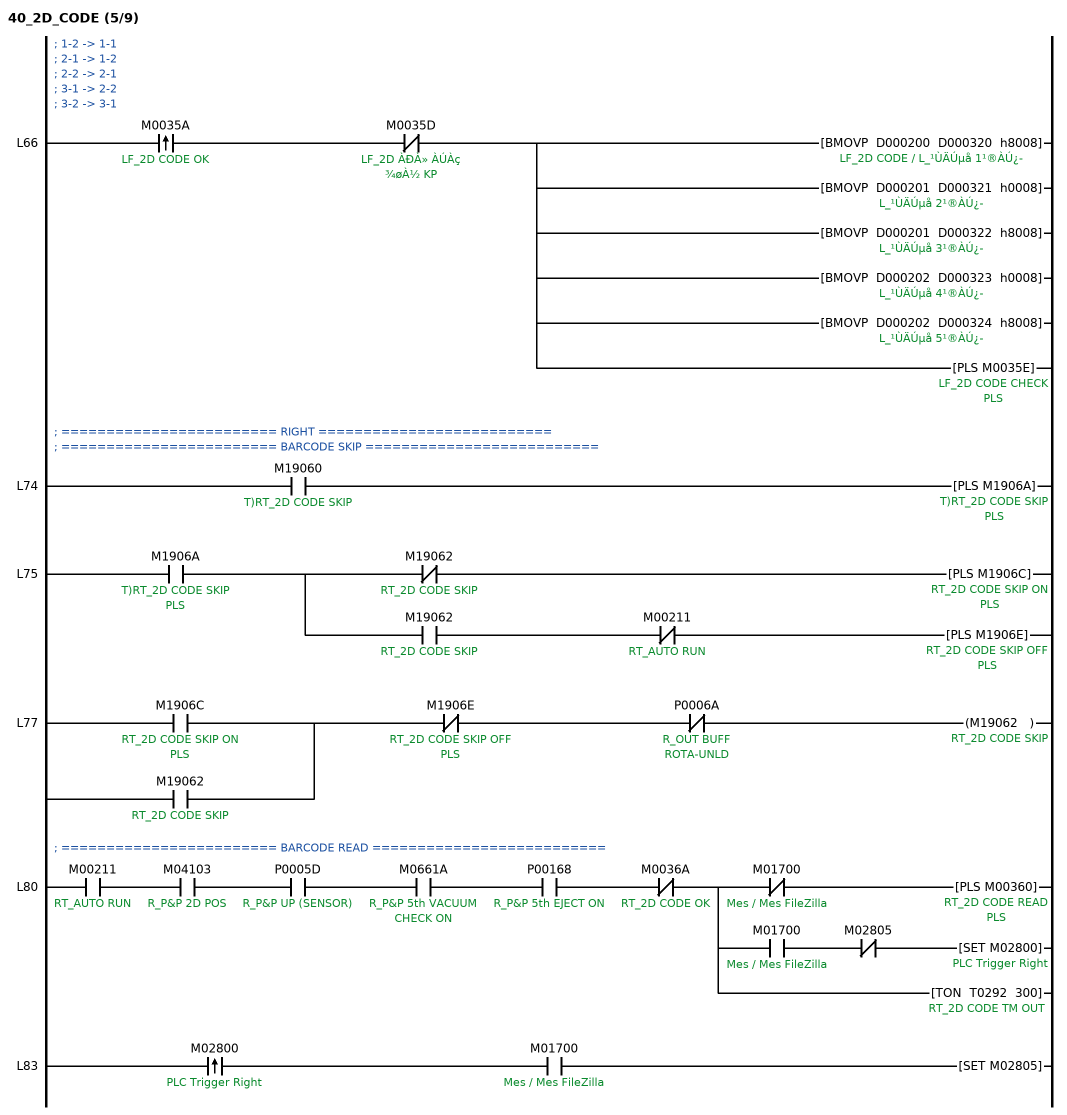
; L66
LOADP     M0035A	// LF_2D CODE OK
AND NOT   M0035D	// LF_2D ÀÐÀ» ÀÚÀç ¾øÀ½ KP
BMOVP     D000200 D000320 h8008	// LF_2D CODE / L_¹ÙÄÚµå 1¹®ÀÚ¿­
BMOVP     D000201 D000321 h0008	// L_¹ÙÄÚµå 2¹®ÀÚ¿­
BMOVP     D000201 D000322 h8008	// L_¹ÙÄÚµå 3¹®ÀÚ¿­
BMOVP     D000202 D000323 h0008	// L_¹ÙÄÚµå 4¹®ÀÚ¿­
BMOVP     D000202 D000324 h8008	// L_¹ÙÄÚµå 5¹®ÀÚ¿­
OUTP      M0035E	// LF_2D CODE CHECK PLS
// output comment: 1-2 -> 1-1
// output comment: 2-1 -> 1-2
// output comment: 2-2 -> 2-1
// output comment: 3-1 -> 2-2
// output comment: 3-2 -> 3-1
// ======================== RIGHT ==========================
// ======================== BARCODE SKIP ==========================
; L74
LOAD      M19060	// T)RT_2D CODE SKIP
OUTP      M1906A	// T)RT_2D CODE SKIP PLS
; L75
LOAD      M1906A	// T)RT_2D CODE SKIP PLS
MPUSH
AND NOT   M19062	// RT_2D CODE SKIP
OUTP      M1906C	// RT_2D CODE SKIP ON PLS
MPOP
AND       M19062	// RT_2D CODE SKIP
AND NOT   M00211	// RT_AUTO RUN
OUTP      M1906E	// RT_2D CODE SKIP OFF PLS
; L77
LOAD      M1906C	// RT_2D CODE SKIP ON PLS
OR        M19062	// RT_2D CODE SKIP
AND NOT   M1906E	// RT_2D CODE SKIP OFF PLS
AND NOT   P0006A	// R_OUT BUFF ROTA-UNLD
OUT       M19062	// RT_2D CODE SKIP
// ======================== BARCODE READ ==========================
; L80
LOAD      M00211	// RT_AUTO RUN
AND       M04103	// R_P&P 2D POS
AND       P0005D	// R_P&P UP (SENSOR)
AND       M0661A	// R_P&P 5th VACUUM CHECK ON
AND       P00168	// R_P&P 5th EJECT ON
AND NOT   M0036A	// RT_2D CODE OK
MPUSH
AND NOT   M01700	// Mes / Mes FileZilla
OUTP      M00360	// RT_2D CODE READ PLS
MLOAD
AND       M01700	// Mes / Mes FileZilla
AND NOT   M02805
SET       M02800	// PLC Trigger Right
MPOP
TON       T0292 300	// RT_2D CODE TM OUT
; L83
LOADP     M02800	// PLC Trigger Right
AND       M01700	// Mes / Mes FileZilla
SET       M02805

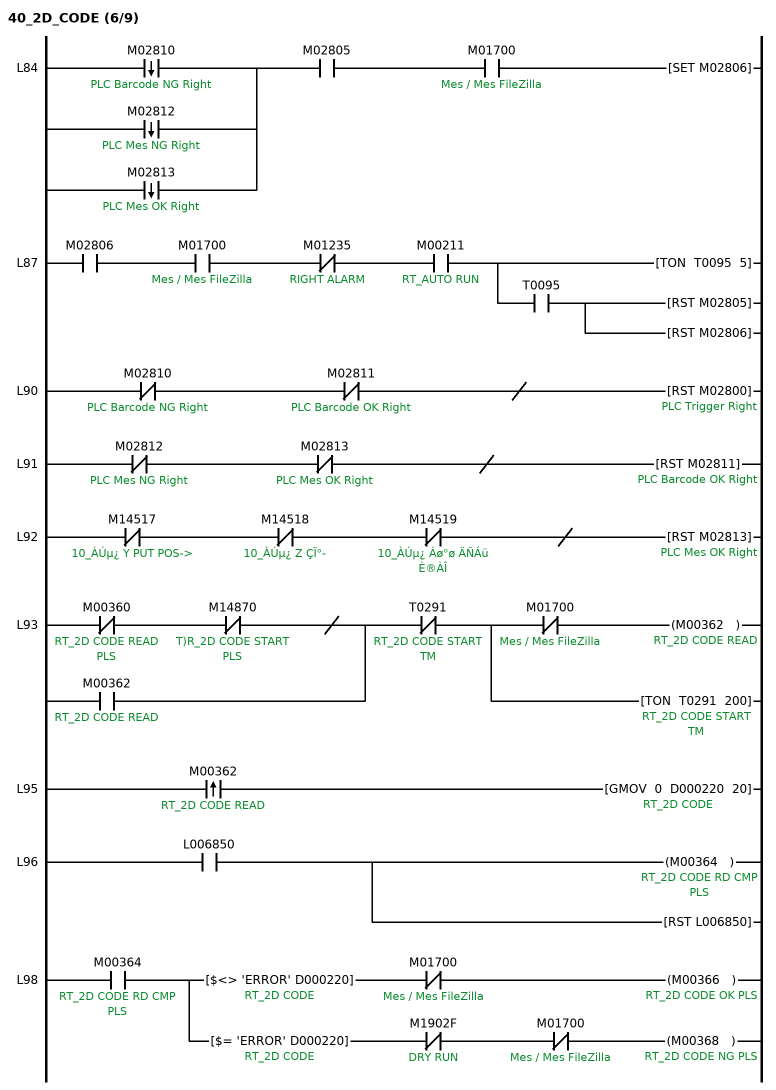
; L84
LOADN     M02810	// PLC Barcode NG Right
ORN       M02812	// PLC Mes NG Right
ORN       M02813	// PLC Mes OK Right
AND       M02805
AND       M01700	// Mes / Mes FileZilla
SET       M02806
; L87
LOAD      M02806
AND       M01700	// Mes / Mes FileZilla
AND NOT   M01235	// RIGHT ALARM
AND       M00211	// RT_AUTO RUN
TON       T0095 5
AND       T0095
RST       M02805
RST       M02806
; L90
LOAD NOT  M02810	// PLC Barcode NG Right
AND NOT   M02811	// PLC Barcode OK Right
NOT
RST       M02800	// PLC Trigger Right
; L91
LOAD NOT  M02812	// PLC Mes NG Right
AND NOT   M02813	// PLC Mes OK Right
NOT
RST       M02811	// PLC Barcode OK Right
; L92
LOAD NOT  M14517	// 10_ÀÚµ¿ Y PUT POS->
AND NOT   M14518	// 10_ÀÚµ¿ Z ÇÏ°­
AND NOT   M14519	// 10_ÀÚµ¿ Áø°ø ÄÑÁü È®ÀÎ
NOT
RST       M02813	// PLC Mes OK Right
; L93
LOAD NOT  M00360	// RT_2D CODE READ PLS
AND NOT   M14870	// T)R_2D CODE START PLS
NOT
OR        M00362	// RT_2D CODE READ
AND NOT   T0291	// RT_2D CODE START TM
MPUSH
AND NOT   M01700	// Mes / Mes FileZilla
OUT       M00362	// RT_2D CODE READ
MPOP
TON       T0291 200	// RT_2D CODE START TM
; L95
LOADP     M00362	// RT_2D CODE READ
GMOV      0 D000220 20	// RT_2D CODE
; L96
LOAD      L006850
OUT       M00364	// RT_2D CODE RD CMP PLS
RST       L006850
; L98
LOAD      M00364	// RT_2D CODE RD CMP PLS
MPUSH
AND$<>    'ERROR' D000220	// RT_2D CODE
AND NOT   M01700	// Mes / Mes FileZilla
OUT       M00366	// RT_2D CODE OK PLS
MPOP
AND$=     'ERROR' D000220	// RT_2D CODE
AND NOT   M1902F	// DRY RUN
AND NOT   M01700	// Mes / Mes FileZilla
OUT       M00368	// RT_2D CODE NG PLS

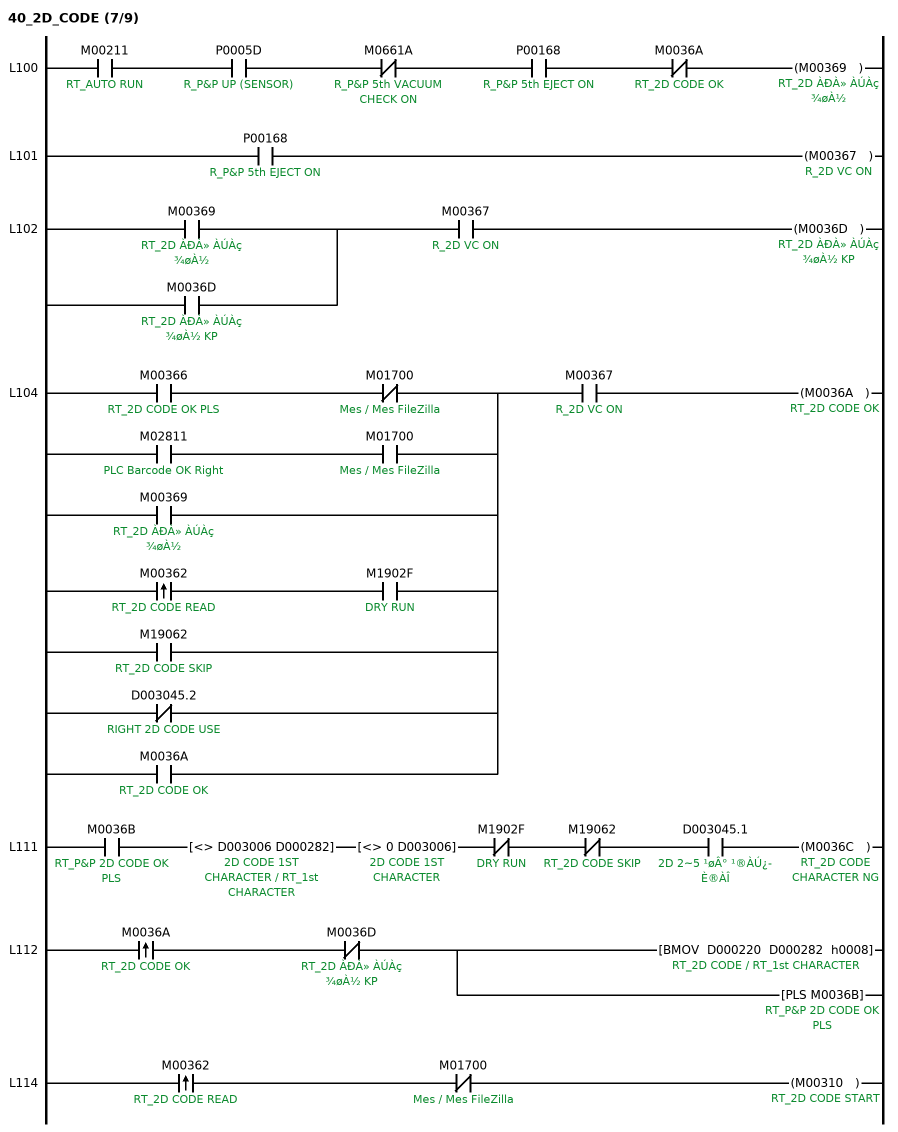
; L100
LOAD      M00211	// RT_AUTO RUN
AND       P0005D	// R_P&P UP (SENSOR)
AND NOT   M0661A	// R_P&P 5th VACUUM CHECK ON
AND       P00168	// R_P&P 5th EJECT ON
AND NOT   M0036A	// RT_2D CODE OK
OUT       M00369	// RT_2D ÀÐÀ» ÀÚÀç ¾øÀ½
; L101
LOAD      P00168	// R_P&P 5th EJECT ON
OUT       M00367	// R_2D VC ON
; L102
LOAD      M00369	// RT_2D ÀÐÀ» ÀÚÀç ¾øÀ½
OR        M0036D	// RT_2D ÀÐÀ» ÀÚÀç ¾øÀ½ KP
AND       M00367	// R_2D VC ON
OUT       M0036D	// RT_2D ÀÐÀ» ÀÚÀç ¾øÀ½ KP
; L104
LOAD      M00366	// RT_2D CODE OK PLS
AND NOT   M01700	// Mes / Mes FileZilla
LOAD      M02811	// PLC Barcode OK Right
AND       M01700	// Mes / Mes FileZilla
OR LOAD
OR        M00369	// RT_2D ÀÐÀ» ÀÚÀç ¾øÀ½
LOADP     M00362	// RT_2D CODE READ
AND       M1902F	// DRY RUN
OR LOAD
OR        M19062	// RT_2D CODE SKIP
OR NOT    D003045.2	// RIGHT 2D CODE USE
OR        M0036A	// RT_2D CODE OK
AND       M00367	// R_2D VC ON
OUT       M0036A	// RT_2D CODE OK
; L111
LOAD      M0036B	// RT_P&P 2D CODE OK PLS
AND<>     D003006 D000282	// 2D CODE 1ST CHARACTER / RT_1st CHARACTER
AND<>     0 D003006	// 2D CODE 1ST CHARACTER
AND NOT   M1902F	// DRY RUN
AND NOT   M19062	// RT_2D CODE SKIP
AND       D003045.1	// 2D 2~5 ¹øÂ° ¹®ÀÚ¿­ È®ÀÎ
OUT       M0036C	// RT_2D CODE CHARACTER NG
; L112
LOADP     M0036A	// RT_2D CODE OK
AND NOT   M0036D	// RT_2D ÀÐÀ» ÀÚÀç ¾øÀ½ KP
BMOV      D000220 D000282 h0008	// RT_2D CODE / RT_1st CHARACTER
OUTP      M0036B	// RT_P&P 2D CODE OK PLS
; L114
LOADP     M00362	// RT_2D CODE READ
AND NOT   M01700	// Mes / Mes FileZilla
OUT       M00310	// RT_2D CODE START

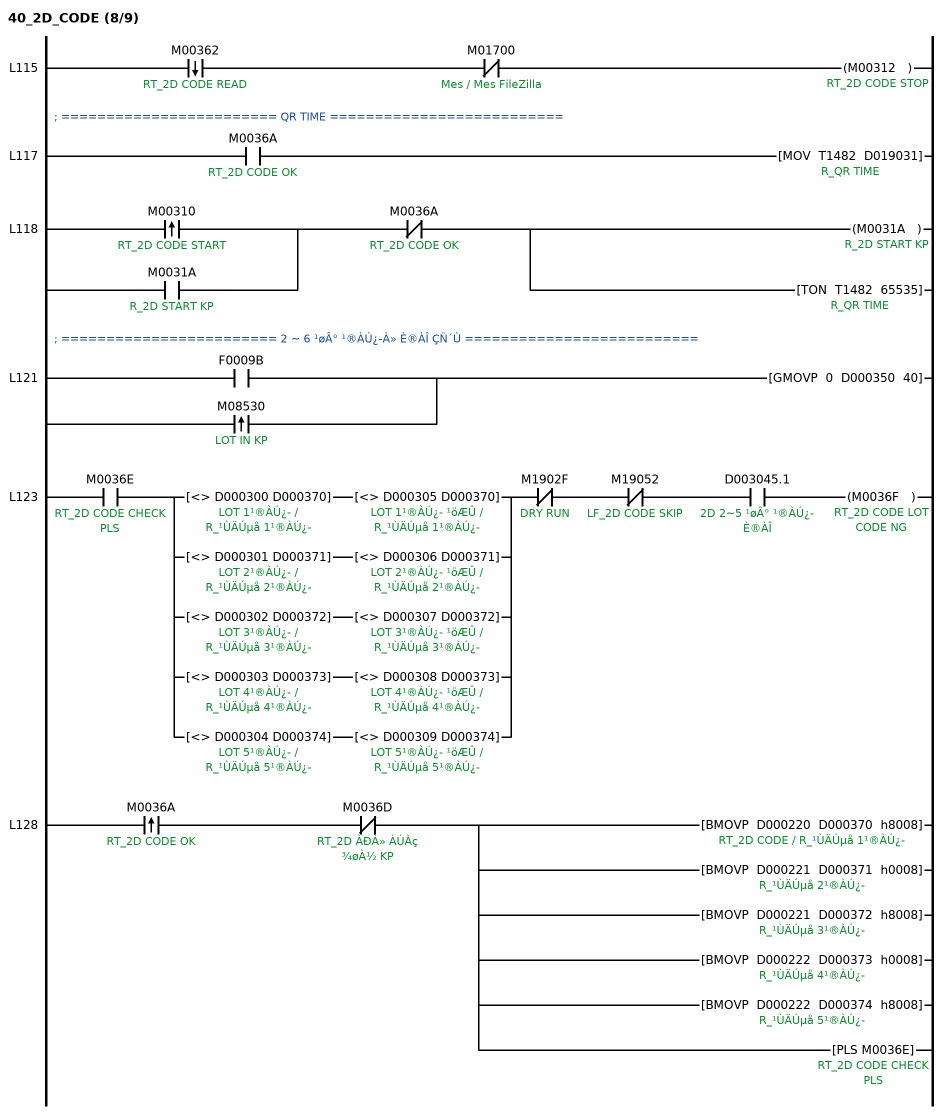
; L115
LOADN     M00362	// RT_2D CODE READ
AND NOT   M01700	// Mes / Mes FileZilla
OUT       M00312	// RT_2D CODE STOP
// ======================== QR TIME ==========================
; L117
LOAD      M0036A	// RT_2D CODE OK
MOV       T1482 D019031	// R_QR TIME
; L118
LOADP     M00310	// RT_2D CODE START
OR        M0031A	// R_2D START KP
AND NOT   M0036A	// RT_2D CODE OK
OUT       M0031A	// R_2D START KP
TON       T1482 65535	// R_QR TIME
// ======================== 2 ~ 6 ¹øÂ° ¹®ÀÚ¿­À» È®ÀÎ ÇÑ´Ù ==========================
; L121
LOAD      F0009B
ORP       M08530	// LOT IN KP
GMOVP     0 D000350 40
; L123
LOAD      M0036E	// RT_2D CODE CHECK PLS
LOAD<>    D000300 D000370	// LOT 1¹®ÀÚ¿­ / R_¹ÙÄÚµå 1¹®ÀÚ¿­
AND<>     D000305 D000370	// LOT 1¹®ÀÚ¿­ ¹öÆÛ / R_¹ÙÄÚµå 1¹®ÀÚ¿­
LOAD<>    D000301 D000371	// LOT 2¹®ÀÚ¿­ / R_¹ÙÄÚµå 2¹®ÀÚ¿­
AND<>     D000306 D000371	// LOT 2¹®ÀÚ¿­ ¹öÆÛ / R_¹ÙÄÚµå 2¹®ÀÚ¿­
OR LOAD
LOAD<>    D000302 D000372	// LOT 3¹®ÀÚ¿­ / R_¹ÙÄÚµå 3¹®ÀÚ¿­
AND<>     D000307 D000372	// LOT 3¹®ÀÚ¿­ ¹öÆÛ / R_¹ÙÄÚµå 3¹®ÀÚ¿­
OR LOAD
LOAD<>    D000303 D000373	// LOT 4¹®ÀÚ¿­ / R_¹ÙÄÚµå 4¹®ÀÚ¿­
AND<>     D000308 D000373	// LOT 4¹®ÀÚ¿­ ¹öÆÛ / R_¹ÙÄÚµå 4¹®ÀÚ¿­
OR LOAD
LOAD<>    D000304 D000374	// LOT 5¹®ÀÚ¿­ / R_¹ÙÄÚµå 5¹®ÀÚ¿­
AND<>     D000309 D000374	// LOT 5¹®ÀÚ¿­ ¹öÆÛ / R_¹ÙÄÚµå 5¹®ÀÚ¿­
OR LOAD
AND LOAD
AND NOT   M1902F	// DRY RUN
AND NOT   M19052	// LF_2D CODE SKIP
AND       D003045.1	// 2D 2~5 ¹øÂ° ¹®ÀÚ¿­ È®ÀÎ
OUT       M0036F	// RT_2D CODE LOT CODE NG
; L128
LOADP     M0036A	// RT_2D CODE OK
AND NOT   M0036D	// RT_2D ÀÐÀ» ÀÚÀç ¾øÀ½ KP
BMOVP     D000220 D000370 h8008	// RT_2D CODE / R_¹ÙÄÚµå 1¹®ÀÚ¿­
BMOVP     D000221 D000371 h0008	// R_¹ÙÄÚµå 2¹®ÀÚ¿­
BMOVP     D000221 D000372 h8008	// R_¹ÙÄÚµå 3¹®ÀÚ¿­
BMOVP     D000222 D000373 h0008	// R_¹ÙÄÚµå 4¹®ÀÚ¿­
BMOVP     D000222 D000374 h8008	// R_¹ÙÄÚµå 5¹®ÀÚ¿­
OUTP      M0036E	// RT_2D CODE CHECK PLS

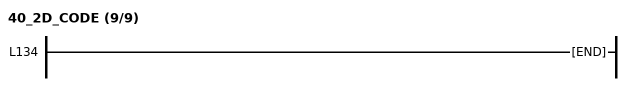
; L134
END

PROGRAM 41_MES (task: ½ºÄµ ÇÁ·Î±×·¥)

